KUKA KRL program: ps_ltc_geo_c2_bolha.src, ps_ltc_geo_c2_bolha.dat

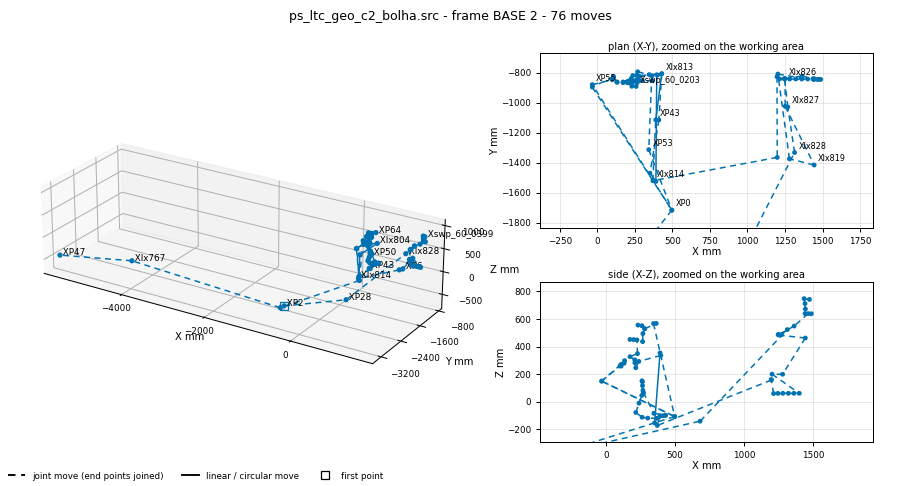
[picture p0: tool path of ps_ltc_geo_c2_bolha.src in frame BASE 2, 76 of 80 moves have a stored position in this frame; points joined in program order, loops and branches not executed]
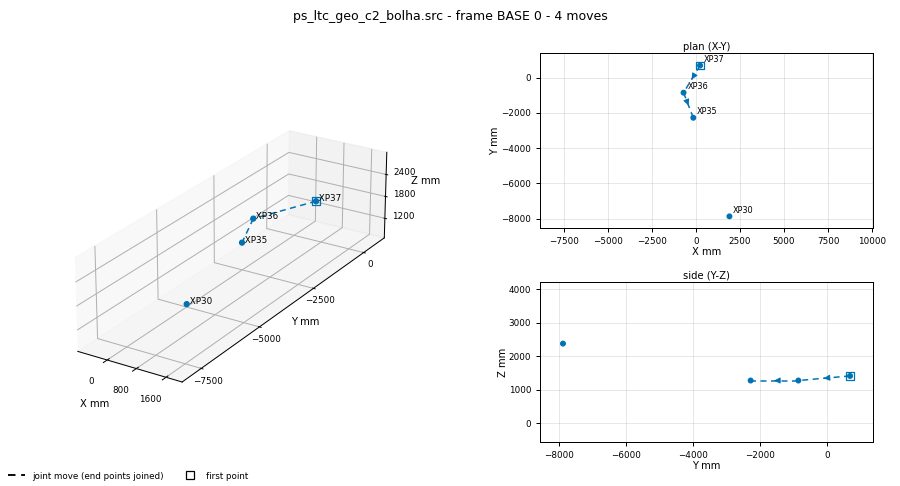
[picture p1: tool path of ps_ltc_geo_c2_bolha.src in frame BASE 0, 4 of 80 moves have a stored position in this frame; points joined in program order, loops and branches not executed]
--- ps_ltc_geo_c2_bolha.src ---
&ACCESS RVO1
&REL 3
&COMMENT GUN C2 geom Accelo
&PARAM DISKPATH = KRC:\R1\Program
DEF ps_ltc_geo_c2_bolha( )
;FOLD INI
;FOLD SPOTTECH INI
USERSPOT(#INIT)
;ENDFOLD (SPOTTECH INI)
;FOLD GRIPPERTECH INI
USER_GRP(0,DUMMY,DUMMY,GDEFAULT)
;ENDFOLD (GRIPPERTECH INI)
  ;FOLD USER INI
    ;Make your modifications here

  ;ENDFOLD (USER INI)
;ENDFOLD (INI)

; Caracterização dos meios de produção:
; Versão Atual:
; 12/07/2013 12:00 Name: P13.050-R3 CHANGES: Solda Geometria Accelo
; Pinça C2

chk_w2_wechs_ok ( )         ; CHECK C2

;FOLD PTP P37 CONT Vel=100 % PDAT38 Tool[2]:Gun C2 Base[2]:Accelo;%{PE}%R 8.2.20,%MKUKATPBASIS,%CMOVE,%VPTP,%P 1:PTP, 2:P37, 3:C_DIS, 5:100, 7:PDAT38
$BWDSTART=FALSE
PDAT_ACT=PPDAT38
FDAT_ACT=FP37
BAS(#PTP_PARAMS,100)
PTP XP37 C_DIS
;ENDFOLD

if MaxStandMenge (2) then
  MaxStandmengeErreicht (2)
endif

IF (NOT(GHOST())) THEN
if Elektrodenwechsel (2) then
  e_fraes2 ()
endif
ENDIF

;FOLD PTP P36 CONT Vel=100 % PDAT37 Tool[2]:Gun C2 Base[2]:Accelo;%{PE}%R 8.2.20,%MKUKATPBASIS,%CMOVE,%VPTP,%P 1:PTP, 2:P36, 3:C_DIS, 5:100, 7:PDAT37
$BWDSTART=FALSE
PDAT_ACT=PPDAT37
FDAT_ACT=FP36
BAS(#PTP_PARAMS,100)
PTP XP36 C_DIS
;ENDFOLD
;FOLD PTP P35 CONT Vel=100 % PDAT36 Tool[2]:Gun C2 Base[2]:Accelo;%{PE}%R 8.2.20,%MKUKATPBASIS,%CMOVE,%VPTP,%P 1:PTP, 2:P35, 3:C_DIS, 5:100, 7:PDAT36
$BWDSTART=FALSE
PDAT_ACT=PPDAT36
FDAT_ACT=FP35
BAS(#PTP_PARAMS,100)
PTP XP35 C_DIS
;ENDFOLD
;FOLD PTP P2 Vel=100 % PDAT2 Tool[2]:Gun C2 Base[2]:Accelo;%{PE}%R 8.2.20,%MKUKATPBASIS,%CMOVE,%VPTP,%P 1:PTP, 2:P2, 3:, 5:100, 7:PDAT2
$BWDSTART=FALSE
PDAT_ACT=PPDAT2
FDAT_ACT=FP2
BAS(#PTP_PARAMS,100)
PTP XP2
;ENDFOLD

;FOLD OUT 3339 'R3 Soldando' State=TRUE ;%{PE}%R 8.2.20,%MKUKATPBASIS,%COUT,%VOUTX,%P 2:3339, 3:R3 Soldando, 5:TRUE, 6:
$OUT[3339]=TRUE
;ENDFOLD
;FOLD WAIT FOR ( IN 3339 'Aguarda Lib. Soldar Geometria' );%{PE}%R 8.2.20,%MKUKATPBASIS,%CEXT_WAIT_FOR,%VEXT_WAIT_FOR,%P 2:, 4:, 5:$IN, 6:3339, 7:Aguarda Lib. Soldar Geometria, 9:
WAIT FOR  ( $IN[3339] )
;ENDFOLD
;FOLD OUT 3339 'R3 Soldando' State=FALSE ;%{PE}%R 8.2.20,%MKUKATPBASIS,%COUT,%VOUTX,%P 2:3339, 3:R3 Soldando, 5:FALSE, 6:
$OUT[3339]=FALSE
;ENDFOLD
;FOLD OUT 3348 'Fora area GEOBOX' State=FALSE ;%{PE}%R 8.2.20,%MKUKATPBASIS,%COUT,%VOUTX,%P 2:3348, 3:Fora area GEOBOX, 5:FALSE, 6:
$OUT[3348]=FALSE
;ENDFOLD

;FOLD Collision.Monitoring_AREA_1_On ;%{PE}%MKUKATPUSER
COLLSTOP( 7, 1 ) ;not Interrupt-Controlled
;ENDFOLD

;FOLD PTP P28 CONT Vel=100 % PDAT28 Tool[2]:Gun C2 Base[2]:Accelo;%{PE}%R 8.2.20,%MKUKATPBASIS,%CMOVE,%VPTP,%P 1:PTP, 2:P28, 3:C_DIS, 5:100, 7:PDAT28
$BWDSTART=FALSE
PDAT_ACT=PPDAT28
FDAT_ACT=FP28
BAS(#PTP_PARAMS,100)
PTP XP28 C_DIS
;ENDFOLD
;FOLD PTP lx828 CONT Vel=100 % P_OLP7 Tool[2]:Gun C2 Base[2]:Accelo;%{PE}%R 8.2.20,%MKUKATPBASIS,%CMOVE,%VPTP,%P 1:PTP, 2:lx828, 3:C_DIS, 5:100, 7:P_OLP7
$BWDSTART=FALSE
PDAT_ACT=PP_OLP7
FDAT_ACT=Flx828
BAS(#PTP_PARAMS,100)
PTP Xlx828 C_DIS
;ENDFOLD
;FOLD PTP lx827 CONT Vel=100 % P_OLP8 Tool[2]:Gun C2 Base[2]:Accelo;%{PE}%R 8.2.20,%MKUKATPBASIS,%CMOVE,%VPTP,%P 1:PTP, 2:lx827, 3:C_DIS, 5:100, 7:P_OLP8
$BWDSTART=FALSE
PDAT_ACT=PP_OLP8
FDAT_ACT=Flx827
BAS(#PTP_PARAMS,100)
PTP Xlx827 C_DIS
;ENDFOLD
;FOLD PTP lx826 CONT Vel=100 % P_OLP9 Tool[2]:Gun C2 Base[2]:Accelo;%{PE}%R 8.2.20,%MKUKATPBASIS,%CMOVE,%VPTP,%P 1:PTP, 2:lx826, 3:C_DIS, 5:100, 7:P_OLP9
$BWDSTART=FALSE
PDAT_ACT=PP_OLP9
FDAT_ACT=Flx826
BAS(#PTP_PARAMS,100)
PTP Xlx826 C_DIS
;ENDFOLD
;FOLD PTP P30 Vel=100 % PDAT30 Tool[2]:Gun C2 Base[0];%{PE}%R 8.2.20,%MKUKATPBASIS,%CMOVE,%VPTP,%P 1:PTP, 2:P30, 3:, 5:100, 7:PDAT30
$BWDSTART=FALSE
PDAT_ACT=PPDAT30
FDAT_ACT=FP30
BAS(#PTP_PARAMS,100)
PTP XP30
;ENDFOLD

;FOLD Collision.Monitoring_AREA_2_On ;%{PE}%MKUKATPUSER
COLLSTOP( 8, 1 ) ;not Interrupt-Controlled
;ENDFOLD

;FOLD ; swp_60_0399;%{PE}%R 5.4.33,%MKUKATPBASIS,%CCOMMENT,%VNORMAL,%P 2:swp_60_0399
;ENDFOLD
;FOLD PTP swp_60_0399 P_OLP10 SPOT Gun=2 RETR CLS PGNO1=110 ACTIVE=1 Tool[2]:Gun C2 Base[2]:Accelo;%{PE}%R 8.2.2,%MKUKATPSPOT,%CSPOT,%VPTP,%P 1:PTP, 2:swp_60_0399, 3:, 5:100, 7:P_OLP10, 10:2, 12:#FIRST, 14:#CLO, 16:151, 18:1, 20:1, 22:0, 24:1, 25:S_OLP1
$BWDSTART=FALSE
PDAT_ACT=PP_OLP10
FDAT_ACT=Fswp_60_0399
BAS(#PTP_PARAMS,PP_OLP10.VEL)
S_ACT.GUN=2
S_ACT.PAIR=SDEFAULT.PAIR
S_ACT.RETR=#CLO
S_ACT.CLO_TM=1
S_ACT.PGNO1=110
S_ACT.PGNO2=SDEFAULT.PGNO2
S_ACT.PRESS1=SDEFAULT.PRESS1
S_ACT.PRESS2=SDEFAULT.PRESS2
S_READY=FALSE
PTP Xswp_60_0399
USERSPOT(#SPOT, S_ACT)
WAIT FOR S_READY
;ENDFOLD

;FOLD PTP P41 CONT Vel=100 % PDAT42 Tool[2]:Gun C2 Base[2]:Accelo;%{PE}%R 8.2.20,%MKUKATPBASIS,%CMOVE,%VPTP,%P 1:PTP, 2:P41, 3:C_DIS, 5:100, 7:PDAT42
$BWDSTART=FALSE
PDAT_ACT=PPDAT42
FDAT_ACT=FP41
BAS(#PTP_PARAMS,100)
PTP XP41 C_DIS
;ENDFOLD


;FOLD ; swp_60_0397;%{PE}%R 8.2.20,%MKUKATPBASIS,%CCOMMENT,%VNORMAL,%P 2:swp_60_0397
;ENDFOLD
;FOLD PTP swp_60_0397 P_OLP15 SPOT Gun=2 RETR CLS PgNo1=145 ACTIVE=1 Tool[2]:Gun C2 Base[2]:Accelo;%{PE}%R 8.2.2,%MKUKATPSPOT,%CSPOT,%VPTP,%P 1:PTP, 2:swp_60_0397, 3:, 5:100, 7:P_OLP15, 10:2, 12:#FIRST, 14:#CLO, 16:145, 18:1, 20:1, 22:0, 24:1, 25:S_OLP2
$BWDSTART=FALSE
PDAT_ACT=PP_OLP15
FDAT_ACT=Fswp_60_0397
BAS(#PTP_PARAMS,PP_OLP15.VEL)
S_ACT.GUN=2
S_ACT.PAIR=SDEFAULT.PAIR
S_ACT.RETR=#CLO
S_ACT.CLO_TM=1
S_ACT.PGNO1=145
S_ACT.PGNO2=SDEFAULT.PGNO2
S_ACT.PRESS1=SDEFAULT.PRESS1
S_ACT.PRESS2=SDEFAULT.PRESS2
S_READY=FALSE
PTP Xswp_60_0397
USERSPOT(#SPOT, S_ACT)
WAIT FOR S_READY
;ENDFOLD

;FOLD ; swp_60_0395;%{PE}%R 5.4.33,%MKUKATPBASIS,%CCOMMENT,%VNORMAL,%P 2:swp_60_0395
;ENDFOLD
;FOLD PTP swp_60_0395 P_OLP12 SPOT Gun=2 RETR CLS PgNo1=111 ACTIVE=1 Tool[2]:Gun C2 Base[2]:Accelo;%{PE}%R 8.2.2,%MKUKATPSPOT,%CSPOT,%VPTP,%P 1:PTP, 2:swp_60_0395, 3:, 5:100, 7:P_OLP12, 10:2, 12:#FIRST, 14:#CLO, 16:111, 18:1, 20:1, 22:0, 24:1, 25:S_OLP2
$BWDSTART=FALSE
PDAT_ACT=PP_OLP12
FDAT_ACT=Fswp_60_0395
BAS(#PTP_PARAMS,PP_OLP12.VEL)
S_ACT.GUN=2
S_ACT.PAIR=SDEFAULT.PAIR
S_ACT.RETR=#CLO
S_ACT.CLO_TM=1
S_ACT.PGNO1=111
S_ACT.PGNO2=SDEFAULT.PGNO2
S_ACT.PRESS1=SDEFAULT.PRESS1
S_ACT.PRESS2=SDEFAULT.PRESS2
S_READY=FALSE
PTP Xswp_60_0395
USERSPOT(#SPOT, S_ACT)
WAIT FOR S_READY
;ENDFOLD

;FOLD PTP lx824 CONT Vel=100 % P_OLP13 Tool[2]:Gun C2 Base[2]:Accelo;%{PE}%R 8.2.20,%MKUKATPBASIS,%CMOVE,%VPTP,%P 1:PTP, 2:lx824, 3:C_DIS, 5:100, 7:P_OLP13
$BWDSTART=FALSE
PDAT_ACT=PP_OLP13
FDAT_ACT=Flx824
BAS(#PTP_PARAMS,100)
PTP Xlx824 C_DIS
;ENDFOLD


;FOLD ; swp_60_0391;%{PE}%R 8.2.20,%MKUKATPBASIS,%CCOMMENT,%VNORMAL,%P 2:swp_60_0391
;ENDFOLD
;FOLD PTP swp_60_0391 P_OLP17 SPOT Gun=2 RETR CLS PgNo1=146 ACTIVE=1 Tool[2]:Gun C2 Base[2]:Accelo;%{PE}%R 8.2.2,%MKUKATPSPOT,%CSPOT,%VPTP,%P 1:PTP, 2:swp_60_0391, 3:, 5:100, 7:P_OLP17, 10:2, 12:#FIRST, 14:#CLO, 16:146, 18:1, 20:1, 22:0, 24:1, 25:S_OLP3
$BWDSTART=FALSE
PDAT_ACT=PP_OLP17
FDAT_ACT=Fswp_60_0391
BAS(#PTP_PARAMS,PP_OLP17.VEL)
S_ACT.GUN=2
S_ACT.PAIR=SDEFAULT.PAIR
S_ACT.RETR=#CLO
S_ACT.CLO_TM=1
S_ACT.PGNO1=146
S_ACT.PGNO2=SDEFAULT.PGNO2
S_ACT.PRESS1=SDEFAULT.PRESS1
S_ACT.PRESS2=SDEFAULT.PRESS2
S_READY=FALSE
PTP Xswp_60_0391
USERSPOT(#SPOT, S_ACT)
WAIT FOR S_READY
;ENDFOLD

;FOLD ; swp_60_0393;%{PE}%R 5.4.33,%MKUKATPBASIS,%CCOMMENT,%VNORMAL,%P 2:swp_60_0393
;ENDFOLD
;FOLD PTP swp_60_0393 P_OLP14 SPOT Gun=2 RETR OPN PGNO1=112 ACTIVE=1 Tool[2]:Gun C2 Base[2]:Accelo;%{PE}%R 8.2.2,%MKUKATPSPOT,%CSPOT,%VPTP,%P 1:PTP, 2:swp_60_0393, 3:, 5:100, 7:P_OLP14, 10:2, 12:#FIRST, 14:#OPN, 16:153, 18:1, 20:1, 22:0, 24:1, 25:S_OLP3
$BWDSTART=FALSE
PDAT_ACT=PP_OLP14
FDAT_ACT=Fswp_60_0393
BAS(#PTP_PARAMS,PP_OLP14.VEL)
S_ACT.GUN=2
S_ACT.PAIR=SDEFAULT.PAIR
S_ACT.RETR=#OPN
S_ACT.CLO_TM=1
S_ACT.PGNO1=112
S_ACT.PGNO2=SDEFAULT.PGNO2
S_ACT.PRESS1=SDEFAULT.PRESS1
S_ACT.PRESS2=SDEFAULT.PRESS2
S_READY=FALSE
PTP Xswp_60_0393
USERSPOT(#SPOT, S_ACT)
WAIT FOR S_READY
;ENDFOLD

;FOLD PTP lx823 CONT Vel=100 % P_OLP16 Tool[2]:Gun C2 Base[2]:Accelo;%{PE}%R 8.2.20,%MKUKATPBASIS,%CMOVE,%VPTP,%P 1:PTP, 2:lx823, 3:C_DIS, 5:100, 7:P_OLP16
$BWDSTART=FALSE
PDAT_ACT=PP_OLP16
FDAT_ACT=Flx823
BAS(#PTP_PARAMS,100)
PTP Xlx823 C_DIS
;ENDFOLD
;FOLD PTP P42 Vel=100 % PDAT43 Tool[2]:Gun C2 Base[2]:Accelo;%{PE}%R 8.2.20,%MKUKATPBASIS,%CMOVE,%VPTP,%P 1:PTP, 2:P42, 3:, 5:100, 7:PDAT43
$BWDSTART=FALSE
PDAT_ACT=PPDAT43
FDAT_ACT=FP42
BAS(#PTP_PARAMS,100)
PTP XP42
;ENDFOLD
;FOLD PTP lx820 Vel=100 % P_OLP18 Tool[2]:Gun C2 Base[2]:Accelo;%{PE}%R 8.2.20,%MKUKATPBASIS,%CMOVE,%VPTP,%P 1:PTP, 2:lx820, 3:, 5:100, 7:P_OLP18
$BWDSTART=FALSE
PDAT_ACT=PP_OLP18
FDAT_ACT=Flx820
BAS(#PTP_PARAMS,100)
PTP Xlx820
;ENDFOLD

;FOLD Collision.Monitoring_AREA_2_Off . ;%{PE}%MKUKATPUSER
COLLSTOP( 8, 2+0 )
;ENDFOLD

;FOLD PTP lx819 CONT Vel=100 % P_OLP19 Tool[2]:Gun C2 Base[2]:Accelo;%{PE}%R 8.2.20,%MKUKATPBASIS,%CMOVE,%VPTP,%P 1:PTP, 2:lx819, 3:C_DIS, 5:100, 7:P_OLP19
$BWDSTART=FALSE
PDAT_ACT=PP_OLP19
FDAT_ACT=Flx819
BAS(#PTP_PARAMS,100)
PTP Xlx819 C_DIS
;ENDFOLD
;FOLD PTP P6 CONT Vel=100 % PDAT6 Tool[2]:Gun C2 Base[2]:Accelo;%{PE}%R 8.2.20,%MKUKATPBASIS,%CMOVE,%VPTP,%P 1:PTP, 2:P6, 3:C_DIS, 5:100, 7:PDAT6
$BWDSTART=FALSE
PDAT_ACT=PPDAT6
FDAT_ACT=FP6
BAS(#PTP_PARAMS,100)
PTP XP6 C_DIS
;ENDFOLD
;FOLD PTP P7 Vel=100 % PDAT7 Tool[2]:Gun C2 Base[2]:Accelo;%{PE}%R 8.2.20,%MKUKATPBASIS,%CMOVE,%VPTP,%P 1:PTP, 2:P7, 3:, 5:100, 7:PDAT7
$BWDSTART=FALSE
PDAT_ACT=PPDAT7
FDAT_ACT=FP7
BAS(#PTP_PARAMS,100)
PTP XP7
;ENDFOLD

;FOLD Collision.Monitoring_AREA_4_On ;%{PE}%MKUKATPUSER
COLLSTOP( 10, 1 ) ;not Interrupt-Controlled
;ENDFOLD

;FOLD ; swp_60_0341;%{PE}%R 8.2.20,%MKUKATPBASIS,%CCOMMENT,%VNORMAL,%P 2:swp_60_0341
;ENDFOLD
;FOLD PTP swp_60_0341 P_OLP21 SPOT Gun=2 RETR CLS PGNO1=113 ACTIVE=1 Tool[2]:Gun C2 Base[2]:Accelo;%{PE}%R 8.2.2,%MKUKATPSPOT,%CSPOT,%VPTP,%P 1:PTP, 2:swp_60_0341, 3:, 5:100, 7:P_OLP21, 10:2, 12:#FIRST, 14:#CLO, 16:154, 18:1, 20:1, 22:0, 24:1, 25:S_OLP4
$BWDSTART=FALSE
PDAT_ACT=PP_OLP21
FDAT_ACT=Fswp_60_0341
BAS(#PTP_PARAMS,PP_OLP21.VEL)
S_ACT.GUN=2
S_ACT.PAIR=SDEFAULT.PAIR
S_ACT.RETR=#CLO
S_ACT.CLO_TM=1
S_ACT.PGNO1=113
S_ACT.PGNO2=SDEFAULT.PGNO2
S_ACT.PRESS1=SDEFAULT.PRESS1
S_ACT.PRESS2=SDEFAULT.PRESS2
S_READY=FALSE
PTP Xswp_60_0341
USERSPOT(#SPOT, S_ACT)
WAIT FOR S_READY
;ENDFOLD

;FOLD ; swp_60_0339;%{PE}%R 8.2.20,%MKUKATPBASIS,%CCOMMENT,%VNORMAL,%P 2:swp_60_0339
;ENDFOLD
;FOLD PTP swp_60_0339 PDAT81 SPOT Gun=2 RETR CLS PGNO1=139 ACTIVE=1 Tool[2]:Gun C2 Base[2]:Accelo;%{PE}%R 8.2.2,%MKUKATPSPOT,%CSPOT,%VPTP,%P 1:PTP, 2:swp_60_0339, 3:, 5:100, 7:PDAT81, 10:2, 12:#FIRST, 14:#CLO, 16:180, 18:1, 20:0, 22:0, 24:1, 25:NORMAL
$BWDSTART=FALSE
PDAT_ACT=PPDAT81
FDAT_ACT=Fswp_60_0339
BAS(#PTP_PARAMS,PPDAT81.VEL)
S_ACT.GUN=2
S_ACT.PAIR=SDEFAULT.PAIR
S_ACT.RETR=#CLO
S_ACT.CLO_TM=1
S_ACT.PGNO1=139
S_ACT.PGNO2=SDEFAULT.PGNO2
S_ACT.PRESS1=SDEFAULT.PRESS1
S_ACT.PRESS2=SDEFAULT.PRESS2
S_READY=FALSE
PTP Xswp_60_0339
USERSPOT(#SPOT, S_ACT)
WAIT FOR S_READY
;ENDFOLD

;FOLD ; swp_60_0337;%{PE}%R 8.2.20,%MKUKATPBASIS,%CCOMMENT,%VNORMAL,%P 2:swp_60_0337
;ENDFOLD
;FOLD PTP swp_60_0337 PDAT82 SPOT Gun=2 RETR CLS PGNO1=140 ACTIVE=1 Tool[2]:Gun C2 Base[2]:Accelo;%{PE}%R 8.2.2,%MKUKATPSPOT,%CSPOT,%VPTP,%P 1:PTP, 2:swp_60_0337, 3:, 5:100, 7:PDAT82, 10:2, 12:#FIRST, 14:#CLO, 16:181, 18:1, 20:0, 22:0, 24:1, 25:NORMAL
$BWDSTART=FALSE
PDAT_ACT=PPDAT82
FDAT_ACT=Fswp_60_0337
BAS(#PTP_PARAMS,PPDAT82.VEL)
S_ACT.GUN=2
S_ACT.PAIR=SDEFAULT.PAIR
S_ACT.RETR=#CLO
S_ACT.CLO_TM=1
S_ACT.PGNO1=140
S_ACT.PGNO2=SDEFAULT.PGNO2
S_ACT.PRESS1=SDEFAULT.PRESS1
S_ACT.PRESS2=SDEFAULT.PRESS2
S_READY=FALSE
PTP Xswp_60_0337
USERSPOT(#SPOT, S_ACT)
WAIT FOR S_READY
;ENDFOLD

;FOLD ; swp_60_0335;%{PE}%R 8.2.20,%MKUKATPBASIS,%CCOMMENT,%VNORMAL,%P 2:swp_60_0335
;ENDFOLD
;FOLD PTP swp_60_0335 PDAT84 SPOT Gun=2 RETR CLS PGNO1=141 ACTIVE=1 Tool[2]:Gun C2 Base[2]:Accelo;%{PE}%R 8.2.2,%MKUKATPSPOT,%CSPOT,%VPTP,%P 1:PTP, 2:swp_60_0335, 3:, 5:100, 7:PDAT84, 10:2, 12:#FIRST, 14:#CLO, 16:182, 18:1, 20:0, 22:0, 24:1, 25:NORMAL
$BWDSTART=FALSE
PDAT_ACT=PPDAT84
FDAT_ACT=Fswp_60_0335
BAS(#PTP_PARAMS,PPDAT84.VEL)
S_ACT.GUN=2
S_ACT.PAIR=SDEFAULT.PAIR
S_ACT.RETR=#CLO
S_ACT.CLO_TM=1
S_ACT.PGNO1=141
S_ACT.PGNO2=SDEFAULT.PGNO2
S_ACT.PRESS1=SDEFAULT.PRESS1
S_ACT.PRESS2=SDEFAULT.PRESS2
S_READY=FALSE
PTP Xswp_60_0335
USERSPOT(#SPOT, S_ACT)
WAIT FOR S_READY
;ENDFOLD

;FOLD ; swp_60_0333;%{PE}%R 8.2.20,%MKUKATPBASIS,%CCOMMENT,%VNORMAL,%P 2:swp_60_0333
;ENDFOLD
;FOLD PTP swp_60_0333 PDAT83 SPOT Gun=2 RETR CLS PGNO1=142 ACTIVE=1 Tool[2]:Gun C2 Base[2]:Accelo;%{PE}%R 8.2.2,%MKUKATPSPOT,%CSPOT,%VPTP,%P 1:PTP, 2:swp_60_0333, 3:, 5:100, 7:PDAT83, 10:2, 12:#FIRST, 14:#CLO, 16:183, 18:1, 20:0, 22:0, 24:1, 25:NORMAL
$BWDSTART=FALSE
PDAT_ACT=PPDAT83
FDAT_ACT=Fswp_60_0333
BAS(#PTP_PARAMS,PPDAT83.VEL)
S_ACT.GUN=2
S_ACT.PAIR=SDEFAULT.PAIR
S_ACT.RETR=#CLO
S_ACT.CLO_TM=1
S_ACT.PGNO1=142
S_ACT.PGNO2=SDEFAULT.PGNO2
S_ACT.PRESS1=SDEFAULT.PRESS1
S_ACT.PRESS2=SDEFAULT.PRESS2
S_READY=FALSE
PTP Xswp_60_0333
USERSPOT(#SPOT, S_ACT)
WAIT FOR S_READY
;ENDFOLD

;FOLD ; swp_60_0331;%{PE}%R 8.2.20,%MKUKATPBASIS,%CCOMMENT,%VNORMAL,%P 2:swp_60_0331
;ENDFOLD
;FOLD PTP swp_60_0331 P_OLP22 SPOT Gun=2 RETR OPN PGNO1=114 ACTIVE=1 Tool[2]:Gun C2 Base[2]:Accelo;%{PE}%R 8.2.2,%MKUKATPSPOT,%CSPOT,%VPTP,%P 1:PTP, 2:swp_60_0331, 3:, 5:100, 7:P_OLP22, 10:2, 12:#FIRST, 14:#OPN, 16:155, 18:1, 20:1, 22:0, 24:1, 25:S_OLP5
$BWDSTART=FALSE
PDAT_ACT=PP_OLP22
FDAT_ACT=Fswp_60_0331
BAS(#PTP_PARAMS,PP_OLP22.VEL)
S_ACT.GUN=2
S_ACT.PAIR=SDEFAULT.PAIR
S_ACT.RETR=#OPN
S_ACT.CLO_TM=1
S_ACT.PGNO1=114
S_ACT.PGNO2=SDEFAULT.PGNO2
S_ACT.PRESS1=SDEFAULT.PRESS1
S_ACT.PRESS2=SDEFAULT.PRESS2
S_READY=FALSE
PTP Xswp_60_0331
USERSPOT(#SPOT, S_ACT)
WAIT FOR S_READY
;ENDFOLD

;FOLD PTP lx815 Vel=100 % P_OLP23 Tool[2]:Gun C2 Base[2]:Accelo;%{PE}%R 8.2.20,%MKUKATPBASIS,%CMOVE,%VPTP,%P 1:PTP, 2:lx815, 3:, 5:100, 7:P_OLP23
$BWDSTART=FALSE
PDAT_ACT=PP_OLP23
FDAT_ACT=Flx815
BAS(#PTP_PARAMS,100)
PTP Xlx815
;ENDFOLD

;FOLD Collision.Monitoring_AREA_4_Off . ;%{PE}%MKUKATPUSER
COLLSTOP( 10, 2+0 )
;ENDFOLD

;FOLD PTP lx816 CONT Vel=100 % P_OLP24 Tool[2]:Gun C2 Base[2]:Accelo;%{PE}%R 8.2.20,%MKUKATPBASIS,%CMOVE,%VPTP,%P 1:PTP, 2:lx816, 3:C_DIS, 5:100, 7:P_OLP24
$BWDSTART=FALSE
PDAT_ACT=PP_OLP24
FDAT_ACT=Flx816
BAS(#PTP_PARAMS,100)
PTP Xlx816 C_DIS
;ENDFOLD
;FOLD PTP lx814 Vel=100 % PDAT35 Tool[2]:Gun C2 Base[2]:Accelo;%{PE}%R 8.2.20,%MKUKATPBASIS,%CMOVE,%VPTP,%P 1:PTP, 2:lx814, 3:, 5:100, 7:PDAT35
$BWDSTART=FALSE
PDAT_ACT=PPDAT35
FDAT_ACT=Flx814
BAS(#PTP_PARAMS,100)
PTP Xlx814
;ENDFOLD

;FOLD Collision.Monitoring_AREA_3_On ;%{PE}%MKUKATPUSER
COLLSTOP( 9, 1 ) ;not Interrupt-Controlled
;ENDFOLD
;FOLD Collision.Monitoring_AREA_1_Off . ;%{PE}%MKUKATPUSER
COLLSTOP( 7, 2+0 )
;ENDFOLD

;FOLD PTP P43 CONT Vel=100 % PDAT85 Tool[2]:Gun C2 Base[2]:Accelo;%{PE}%R 8.2.20,%MKUKATPBASIS,%CMOVE,%VPTP,%P 1:PTP, 2:P43, 3:C_DIS, 5:100, 7:PDAT85
$BWDSTART=FALSE
PDAT_ACT=PPDAT85
FDAT_ACT=FP43
BAS(#PTP_PARAMS,100)
PTP XP43 C_DIS
;ENDFOLD

;FOLD LIN lx813 CONT Vel=1 m/s CPDAT5 Tool[2]:Gun C2 Base[2]:Accelo;%{PE}%R 8.2.20,%MKUKATPBASIS,%CMOVE,%VLIN,%P 1:LIN, 2:lx813, 3:C_DIS C_DIS, 5:1, 7:CPDAT5
$BWDSTART=FALSE
LDAT_ACT=LCPDAT5
FDAT_ACT=Flx813
BAS(#CP_PARAMS,1)
LIN Xlx813 C_DIS C_DIS
;ENDFOLD

;FOLD ; swp_60_0259;%{PE}%R 8.2.20,%MKUKATPBASIS,%CCOMMENT,%VNORMAL,%P 2:swp_60_0259
;ENDFOLD
;FOLD PTP swp_60_0259 PDAT55 SPOT Gun=2 RETR CLS PGNO1=96 ACTIVE=1 Tool[2]:Gun C2 Base[2]:Accelo;%{PE}%R 8.2.2,%MKUKATPSPOT,%CSPOT,%VPTP,%P 1:PTP, 2:swp_60_0259, 3:, 5:100, 7:PDAT55, 10:2, 12:#FIRST, 14:#CLO, 16:137, 18:1, 20:0, 22:0, 24:1, 25:NORMAL
$BWDSTART=FALSE
PDAT_ACT=PPDAT55
FDAT_ACT=Fswp_60_0259
BAS(#PTP_PARAMS,PPDAT55.VEL)
S_ACT.GUN=2
S_ACT.PAIR=SDEFAULT.PAIR
S_ACT.RETR=#CLO
S_ACT.CLO_TM=1
S_ACT.PGNO1=96
S_ACT.PGNO2=SDEFAULT.PGNO2
S_ACT.PRESS1=SDEFAULT.PRESS1
S_ACT.PRESS2=SDEFAULT.PRESS2
S_READY=FALSE
PTP Xswp_60_0259
USERSPOT(#SPOT, S_ACT)
WAIT FOR S_READY
;ENDFOLD

;FOLD ; swp_60_0255;%{PE}%R 5.4.33,%MKUKATPBASIS,%CCOMMENT,%VNORMAL,%P 2:swp_60_0255
;ENDFOLD
;FOLD PTP swp_60_0255 P_OLP30 SPOT Gun=2 RETR CLS PGNO1=115 ACTIVE=1 Tool[2]:Gun C2 Base[2]:Accelo;%{PE}%R 8.2.2,%MKUKATPSPOT,%CSPOT,%VPTP,%P 1:PTP, 2:swp_60_0255, 3:, 5:100, 7:P_OLP30, 10:2, 12:#FIRST, 14:#CLO, 16:156, 18:1, 20:1, 22:0, 24:1, 25:S_OLP6
$BWDSTART=FALSE
PDAT_ACT=PP_OLP30
FDAT_ACT=Fswp_60_0255
BAS(#PTP_PARAMS,PP_OLP30.VEL)
S_ACT.GUN=2
S_ACT.PAIR=SDEFAULT.PAIR
S_ACT.RETR=#CLO
S_ACT.CLO_TM=1
S_ACT.PGNO1=115
S_ACT.PGNO2=SDEFAULT.PGNO2
S_ACT.PRESS1=SDEFAULT.PRESS1
S_ACT.PRESS2=SDEFAULT.PRESS2
S_READY=FALSE
PTP Xswp_60_0255
USERSPOT(#SPOT, S_ACT)
WAIT FOR S_READY
;ENDFOLD

;FOLD ; swp_60_0253;%{PE}%R 8.2.20,%MKUKATPBASIS,%CCOMMENT,%VNORMAL,%P 2:swp_60_0253
;ENDFOLD
;FOLD PTP swp_60_0253 PDAT56 SPOT Gun=2 RETR CLS PGNO1=94 ACTIVE=1 Tool[2]:Gun C2 Base[2]:Accelo;%{PE}%R 8.2.2,%MKUKATPSPOT,%CSPOT,%VPTP,%P 1:PTP, 2:swp_60_0253, 3:, 5:100, 7:PDAT56, 10:2, 12:#FIRST, 14:#CLO, 16:135, 18:1, 20:0, 22:0, 24:1, 25:NORMAL
$BWDSTART=FALSE
PDAT_ACT=PPDAT56
FDAT_ACT=Fswp_60_0253
BAS(#PTP_PARAMS,PPDAT56.VEL)
S_ACT.GUN=2
S_ACT.PAIR=SDEFAULT.PAIR
S_ACT.RETR=#CLO
S_ACT.CLO_TM=1
S_ACT.PGNO1=94
S_ACT.PGNO2=SDEFAULT.PGNO2
S_ACT.PRESS1=SDEFAULT.PRESS1
S_ACT.PRESS2=SDEFAULT.PRESS2
S_READY=FALSE
PTP Xswp_60_0253
USERSPOT(#SPOT, S_ACT)
WAIT FOR S_READY
;ENDFOLD

;FOLD ; swp_60_0249;%{PE}%R 8.2.20,%MKUKATPBASIS,%CCOMMENT,%VNORMAL,%P 2:swp_60_0249
;ENDFOLD
;FOLD PTP swp_60_0249 PDAT57 SPOT Gun=2 RETR CLS PGNO1=92 ACTIVE=1 Tool[2]:Gun C2 Base[2]:Accelo;%{PE}%R 8.2.2,%MKUKATPSPOT,%CSPOT,%VPTP,%P 1:PTP, 2:swp_60_0249, 3:, 5:100, 7:PDAT57, 10:2, 12:#FIRST, 14:#CLO, 16:133, 18:1, 20:0, 22:0, 24:1, 25:NORMAL
$BWDSTART=FALSE
PDAT_ACT=PPDAT57
FDAT_ACT=Fswp_60_0249
BAS(#PTP_PARAMS,PPDAT57.VEL)
S_ACT.GUN=2
S_ACT.PAIR=SDEFAULT.PAIR
S_ACT.RETR=#CLO
S_ACT.CLO_TM=1
S_ACT.PGNO1=92
S_ACT.PGNO2=SDEFAULT.PGNO2
S_ACT.PRESS1=SDEFAULT.PRESS1
S_ACT.PRESS2=SDEFAULT.PRESS2
S_READY=FALSE
PTP Xswp_60_0249
USERSPOT(#SPOT, S_ACT)
WAIT FOR S_READY
;ENDFOLD

;FOLD ; swp_60_0245;%{PE}%R 5.4.33,%MKUKATPBASIS,%CCOMMENT,%VNORMAL,%P 2:swp_60_0245
;ENDFOLD
;FOLD PTP swp_60_0245 P_OLP31 SPOT Gun=2 RETR CLS PGNO1=116 ACTIVE=1 Tool[2]:Gun C2 Base[2]:Accelo;%{PE}%R 8.2.2,%MKUKATPSPOT,%CSPOT,%VPTP,%P 1:PTP, 2:swp_60_0245, 3:, 5:100, 7:P_OLP31, 10:2, 12:#FIRST, 14:#CLO, 16:157, 18:1, 20:1, 22:0, 24:1, 25:S_OLP7
$BWDSTART=FALSE
PDAT_ACT=PP_OLP31
FDAT_ACT=Fswp_60_0245
BAS(#PTP_PARAMS,PP_OLP31.VEL)
S_ACT.GUN=2
S_ACT.PAIR=SDEFAULT.PAIR
S_ACT.RETR=#CLO
S_ACT.CLO_TM=1
S_ACT.PGNO1=116
S_ACT.PGNO2=SDEFAULT.PGNO2
S_ACT.PRESS1=SDEFAULT.PRESS1
S_ACT.PRESS2=SDEFAULT.PRESS2
S_READY=FALSE
PTP Xswp_60_0245
USERSPOT(#SPOT, S_ACT)
WAIT FOR S_READY
;ENDFOLD

;FOLD ; swp_60_0241;%{PE}%R 8.2.20,%MKUKATPBASIS,%CCOMMENT,%VNORMAL,%P 2:swp_60_0241
;ENDFOLD
;FOLD PTP swp_60_0241 PDAT58 SPOT Gun=2 RETR CLS PGNO1=89 ACTIVE=1 Tool[2]:Gun C2 Base[2]:Accelo;%{PE}%R 8.2.2,%MKUKATPSPOT,%CSPOT,%VPTP,%P 1:PTP, 2:swp_60_0241, 3:, 5:100, 7:PDAT58, 10:2, 12:#FIRST, 14:#CLO, 16:130, 18:1, 20:0, 22:0, 24:1, 25:NORMAL
$BWDSTART=FALSE
PDAT_ACT=PPDAT58
FDAT_ACT=Fswp_60_0241
BAS(#PTP_PARAMS,PPDAT58.VEL)
S_ACT.GUN=2
S_ACT.PAIR=SDEFAULT.PAIR
S_ACT.RETR=#CLO
S_ACT.CLO_TM=1
S_ACT.PGNO1=89
S_ACT.PGNO2=SDEFAULT.PGNO2
S_ACT.PRESS1=SDEFAULT.PRESS1
S_ACT.PRESS2=SDEFAULT.PRESS2
S_READY=FALSE
PTP Xswp_60_0241
USERSPOT(#SPOT, S_ACT)
WAIT FOR S_READY
;ENDFOLD

;FOLD PTP P50 CONT Vel=100 % PDAT59 Tool[2]:Gun C2 Base[2]:Accelo;%{PE}%R 8.2.20,%MKUKATPBASIS,%CMOVE,%VPTP,%P 1:PTP, 2:P50, 3:C_DIS, 5:100, 7:PDAT59
$BWDSTART=FALSE
PDAT_ACT=PPDAT59
FDAT_ACT=FP50
BAS(#PTP_PARAMS,100)
PTP XP50 C_DIS
;ENDFOLD

;FOLD ; swp_60_0239;%{PE}%R 8.2.20,%MKUKATPBASIS,%CCOMMENT,%VNORMAL,%P 2:swp_60_0239
;ENDFOLD
;FOLD PTP swp_60_0239 PDAT60 SPOT Gun=2 RETR CLS PGNO1=88 ACTIVE=1 Tool[2]:Gun C2 Base[2]:Accelo;%{PE}%R 8.2.2,%MKUKATPSPOT,%CSPOT,%VPTP,%P 1:PTP, 2:swp_60_0239, 3:, 5:100, 7:PDAT60, 10:2, 12:#FIRST, 14:#CLO, 16:129, 18:1, 20:0, 22:0, 24:1, 25:NORMAL
$BWDSTART=FALSE
PDAT_ACT=PPDAT60
FDAT_ACT=Fswp_60_0239
BAS(#PTP_PARAMS,PPDAT60.VEL)
S_ACT.GUN=2
S_ACT.PAIR=SDEFAULT.PAIR
S_ACT.RETR=#CLO
S_ACT.CLO_TM=1
S_ACT.PGNO1=88
S_ACT.PGNO2=SDEFAULT.PGNO2
S_ACT.PRESS1=SDEFAULT.PRESS1
S_ACT.PRESS2=SDEFAULT.PRESS2
S_READY=FALSE
PTP Xswp_60_0239
USERSPOT(#SPOT, S_ACT)
WAIT FOR S_READY
;ENDFOLD

;FOLD ; swp_60_0237;%{PE}%R 8.2.20,%MKUKATPBASIS,%CCOMMENT,%VNORMAL,%P 2:swp_60_0237
;ENDFOLD
;FOLD PTP swp_60_0237 PDAT61 SPOT Gun=2 RETR CLS PGNO1=87 ACTIVE=1 Tool[2]:Gun C2 Base[2]:Accelo;%{PE}%R 8.2.2,%MKUKATPSPOT,%CSPOT,%VPTP,%P 1:PTP, 2:swp_60_0237, 3:, 5:100, 7:PDAT61, 10:2, 12:#FIRST, 14:#CLO, 16:128, 18:1, 20:0, 22:0, 24:1, 25:NORMAL
$BWDSTART=FALSE
PDAT_ACT=PPDAT61
FDAT_ACT=Fswp_60_0237
BAS(#PTP_PARAMS,PPDAT61.VEL)
S_ACT.GUN=2
S_ACT.PAIR=SDEFAULT.PAIR
S_ACT.RETR=#CLO
S_ACT.CLO_TM=1
S_ACT.PGNO1=87
S_ACT.PGNO2=SDEFAULT.PGNO2
S_ACT.PRESS1=SDEFAULT.PRESS1
S_ACT.PRESS2=SDEFAULT.PRESS2
S_READY=FALSE
PTP Xswp_60_0237
USERSPOT(#SPOT, S_ACT)
WAIT FOR S_READY
;ENDFOLD

;FOLD PTP P11 CONT Vel=50 % PDAT11 Tool[2]:Gun C2 Base[2]:Accelo;%{PE}%R 8.2.20,%MKUKATPBASIS,%CMOVE,%VPTP,%P 1:PTP, 2:P11, 3:C_DIS, 5:50, 7:PDAT11
$BWDSTART=FALSE
PDAT_ACT=PPDAT11
FDAT_ACT=FP11
BAS(#PTP_PARAMS,50)
PTP XP11 C_DIS
;ENDFOLD

;FOLD ; swp_60_0235;%{PE}%R 5.4.33,%MKUKATPBASIS,%CCOMMENT,%VNORMAL,%P 2:swp_60_0235
;ENDFOLD
;FOLD PTP swp_60_0235 P_OLP33 SPOT Gun=2 RETR OPN PGNO1=117 ACTIVE=1 Tool[2]:Gun C2 Base[2]:Accelo;%{PE}%R 8.2.2,%MKUKATPSPOT,%CSPOT,%VPTP,%P 1:PTP, 2:swp_60_0235, 3:, 5:100, 7:P_OLP33, 10:2, 12:#FIRST, 14:#OPN, 16:158, 18:1, 20:1, 22:0, 24:1, 25:S_OLP8
$BWDSTART=FALSE
PDAT_ACT=PP_OLP33
FDAT_ACT=Fswp_60_0235
BAS(#PTP_PARAMS,PP_OLP33.VEL)
S_ACT.GUN=2
S_ACT.PAIR=SDEFAULT.PAIR
S_ACT.RETR=#OPN
S_ACT.CLO_TM=1
S_ACT.PGNO1=117
S_ACT.PGNO2=SDEFAULT.PGNO2
S_ACT.PRESS1=SDEFAULT.PRESS1
S_ACT.PRESS2=SDEFAULT.PRESS2
S_READY=FALSE
PTP Xswp_60_0235
USERSPOT(#SPOT, S_ACT)
WAIT FOR S_READY
;ENDFOLD

;FOLD PTP lx798 CONT Vel=100 % P_OLP34 Tool[2]:Gun C2 Base[2]:Accelo;%{PE}%R 8.2.20,%MKUKATPBASIS,%CMOVE,%VPTP,%P 1:PTP, 2:lx798, 3:C_DIS, 5:100, 7:P_OLP34
$BWDSTART=FALSE
PDAT_ACT=PP_OLP34
FDAT_ACT=Flx798
BAS(#PTP_PARAMS,100)
PTP Xlx798 C_DIS
;ENDFOLD
;FOLD PTP lx799 CONT Vel=100 % P_OLP35 Tool[2]:Gun C2 Base[2]:Accelo;%{PE}%R 8.2.20,%MKUKATPBASIS,%CMOVE,%VPTP,%P 1:PTP, 2:lx799, 3:C_DIS, 5:100, 7:P_OLP35
$BWDSTART=FALSE
PDAT_ACT=PP_OLP35
FDAT_ACT=Flx799
BAS(#PTP_PARAMS,100)
PTP Xlx799 C_DIS
;ENDFOLD

;FOLD LIN lx800 CONT Vel=1 m/s CPDAT8 Tool[2]:Gun C2 Base[2]:Accelo;%{PE}%R 8.2.20,%MKUKATPBASIS,%CMOVE,%VLIN,%P 1:LIN, 2:lx800, 3:C_DIS C_DIS, 5:1, 7:CPDAT8
$BWDSTART=FALSE
LDAT_ACT=LCPDAT8
FDAT_ACT=Flx800
BAS(#CP_PARAMS,1)
LIN Xlx800 C_DIS C_DIS
;ENDFOLD

;FOLD PTP lx802 CONT Vel=100 % P_OLP37 Tool[2]:Gun C2 Base[2]:Accelo;%{PE}%R 8.2.20,%MKUKATPBASIS,%CMOVE,%VPTP,%P 1:PTP, 2:lx802, 3:C_DIS, 5:100, 7:P_OLP37
$BWDSTART=FALSE
PDAT_ACT=PP_OLP37
FDAT_ACT=Flx802
BAS(#PTP_PARAMS,100)
PTP Xlx802 C_DIS
;ENDFOLD
;FOLD PTP lx801 CONT Vel=100 % P_OLP38 Tool[2]:Gun C2 Base[2]:Accelo;%{PE}%R 8.2.20,%MKUKATPBASIS,%CMOVE,%VPTP,%P 1:PTP, 2:lx801, 3:C_DIS, 5:100, 7:P_OLP38
$BWDSTART=FALSE
PDAT_ACT=PP_OLP38
FDAT_ACT=Flx801
BAS(#PTP_PARAMS,100)
PTP Xlx801 C_DIS
;ENDFOLD

;FOLD LIN P62 CONT Vel=1.5 m/s CPDAT11 Tool[2]:Gun C2 Base[2]:Accelo;%{PE}%R 8.2.20,%MKUKATPBASIS,%CMOVE,%VLIN,%P 1:LIN, 2:P62, 3:C_DIS C_DIS, 5:1.5, 7:CPDAT11
$BWDSTART=FALSE
LDAT_ACT=LCPDAT11
FDAT_ACT=FP62
BAS(#CP_PARAMS,1.5)
LIN XP62 C_DIS C_DIS
;ENDFOLD
;FOLD LIN lx804 CONT Vel=1 m/s CPDAT1 Tool[2]:Gun C2 Base[2]:Accelo;%{PE}%R 8.2.20,%MKUKATPBASIS,%CMOVE,%VLIN,%P 1:LIN, 2:lx804, 3:C_DIS C_DIS, 5:1, 7:CPDAT1
$BWDSTART=FALSE
LDAT_ACT=LCPDAT1
FDAT_ACT=Flx804
BAS(#CP_PARAMS,1)
LIN Xlx804 C_DIS C_DIS
;ENDFOLD

;FOLD PTP lx803 CONT Vel=100 % P_OLP45 Tool[2]:Gun C2 Base[2]:Accelo;%{PE}%R 8.2.20,%MKUKATPBASIS,%CMOVE,%VPTP,%P 1:PTP, 2:lx803, 3:C_DIS, 5:100, 7:P_OLP45
$BWDSTART=FALSE
PDAT_ACT=PP_OLP45
FDAT_ACT=Flx803
BAS(#PTP_PARAMS,100)
PTP Xlx803 C_DIS
;ENDFOLD

;FOLD ; swp_60_0229;%{PE}%R 5.4.33,%MKUKATPBASIS,%CCOMMENT,%VNORMAL,%P 2:swp_60_0229
;ENDFOLD
;FOLD PTP swp_60_0229 P_OLP46 SPOT Gun=2 RETR CLS PGNO1=118 ACTIVE=1 Tool[2]:Gun C2 Base[2]:Accelo;%{PE}%R 8.2.2,%MKUKATPSPOT,%CSPOT,%VPTP,%P 1:PTP, 2:swp_60_0229, 3:, 5:100, 7:P_OLP46, 10:2, 12:#FIRST, 14:#CLO, 16:159, 18:1, 20:1, 22:0, 24:1, 25:S_OLP9
$BWDSTART=FALSE
PDAT_ACT=PP_OLP46
FDAT_ACT=Fswp_60_0229
BAS(#PTP_PARAMS,PP_OLP46.VEL)
S_ACT.GUN=2
S_ACT.PAIR=SDEFAULT.PAIR
S_ACT.RETR=#CLO
S_ACT.CLO_TM=1
S_ACT.PGNO1=118
S_ACT.PGNO2=SDEFAULT.PGNO2
S_ACT.PRESS1=SDEFAULT.PRESS1
S_ACT.PRESS2=SDEFAULT.PRESS2
S_READY=FALSE
PTP Xswp_60_0229
USERSPOT(#SPOT, S_ACT)
WAIT FOR S_READY
;ENDFOLD

;FOLD ; swp_60_0225;%{PE}%R 5.4.33,%MKUKATPBASIS,%CCOMMENT,%VNORMAL,%P 2:swp_60_0225
;ENDFOLD
;FOLD PTP swp_60_0225 P_OLP47 SPOT Gun=2 RETR CLS PGNO1=119 ACTIVE=1 Tool[2]:Gun C2 Base[2]:Accelo;%{PE}%R 8.2.2,%MKUKATPSPOT,%CSPOT,%VPTP,%P 1:PTP, 2:swp_60_0225, 3:, 5:100, 7:P_OLP47, 10:2, 12:#FIRST, 14:#CLO, 16:160, 18:1, 20:1, 22:0, 24:1, 25:S_OLP10
$BWDSTART=FALSE
PDAT_ACT=PP_OLP47
FDAT_ACT=Fswp_60_0225
BAS(#PTP_PARAMS,PP_OLP47.VEL)
S_ACT.GUN=2
S_ACT.PAIR=SDEFAULT.PAIR
S_ACT.RETR=#CLO
S_ACT.CLO_TM=1
S_ACT.PGNO1=119
S_ACT.PGNO2=SDEFAULT.PGNO2
S_ACT.PRESS1=SDEFAULT.PRESS1
S_ACT.PRESS2=SDEFAULT.PRESS2
S_READY=FALSE
PTP Xswp_60_0225
USERSPOT(#SPOT, S_ACT)
WAIT FOR S_READY
;ENDFOLD

;FOLD PTP PS01010021 PDAT86 RETR OPN Gun=2 Tool[2]:Gun C2 Base[2]:Accelo;%{PE}%R 8.2.2,%MKUKATPSPOT,%CRETR,%VPTP,%P 1:PTP, 2:PS01010021, 3:, 5:100, 7:PDAT86, 9:#OPN, 11:2, 13:#FIRST
$BWDSTART=FALSE
PDAT_ACT=PPDAT86
FDAT_ACT=FPS01010021
BAS(#PTP_PARAMS,PPDAT86.VEL)
S_ACT.GUN=2
S_ACT.PAIR=#FIRST
S_ACT.RETR=#OPN
S_READY=FALSE
PTP XPS01010021
USERSPOT(#RETR, S_ACT)
WAIT FOR S_READY
;ENDFOLD

;FOLD ; swp_60_0221;%{PE}%R 5.4.33,%MKUKATPBASIS,%CCOMMENT,%VNORMAL,%P 2:swp_60_0221
;ENDFOLD
;FOLD PTP swp_60_0221 P_OLP49 SPOT Gun=2 RETR OPN PGNO1=120 ACTIVE=1 Tool[2]:Gun C2 Base[2]:Accelo;%{PE}%R 8.2.2,%MKUKATPSPOT,%CSPOT,%VPTP,%P 1:PTP, 2:swp_60_0221, 3:, 5:100, 7:P_OLP49, 10:2, 12:#FIRST, 14:#OPN, 16:161, 18:1, 20:1, 22:0, 24:1, 25:S_OLP11
$BWDSTART=FALSE
PDAT_ACT=PP_OLP49
FDAT_ACT=Fswp_60_0221
BAS(#PTP_PARAMS,PP_OLP49.VEL)
S_ACT.GUN=2
S_ACT.PAIR=SDEFAULT.PAIR
S_ACT.RETR=#OPN
S_ACT.CLO_TM=1
S_ACT.PGNO1=120
S_ACT.PGNO2=SDEFAULT.PGNO2
S_ACT.PRESS1=SDEFAULT.PRESS1
S_ACT.PRESS2=SDEFAULT.PRESS2
S_READY=FALSE
PTP Xswp_60_0221
USERSPOT(#SPOT, S_ACT)
WAIT FOR S_READY
;ENDFOLD

;FOLD PTP lx795 CONT Vel=100 % P_OLP50 Tool[2]:Gun C2 Base[2]:Accelo;%{PE}%R 8.2.20,%MKUKATPBASIS,%CMOVE,%VPTP,%P 1:PTP, 2:lx795, 3:C_DIS, 5:100, 7:P_OLP50
$BWDSTART=FALSE
PDAT_ACT=PP_OLP50
FDAT_ACT=Flx795
BAS(#PTP_PARAMS,100)
PTP Xlx795 C_DIS
;ENDFOLD

;FOLD ; swp_60_0207;%{PE}%R 8.2.20,%MKUKATPBASIS,%CCOMMENT,%VNORMAL,%P 2:swp_60_0207
;ENDFOLD
;FOLD PTP swp_60_0207 PDAT62 SPOT Gun=2 RETR CLS PGNO1=81 ACTIVE=1 Tool[2]:Gun C2 Base[2]:Accelo;%{PE}%R 8.2.2,%MKUKATPSPOT,%CSPOT,%VPTP,%P 1:PTP, 2:swp_60_0207, 3:, 5:100, 7:PDAT62, 10:2, 12:#FIRST, 14:#CLO, 16:122, 18:1, 20:0, 22:0, 24:1, 25:NORMAL
$BWDSTART=FALSE
PDAT_ACT=PPDAT62
FDAT_ACT=Fswp_60_0207
BAS(#PTP_PARAMS,PPDAT62.VEL)
S_ACT.GUN=2
S_ACT.PAIR=SDEFAULT.PAIR
S_ACT.RETR=#CLO
S_ACT.CLO_TM=1
S_ACT.PGNO1=81
S_ACT.PGNO2=SDEFAULT.PGNO2
S_ACT.PRESS1=SDEFAULT.PRESS1
S_ACT.PRESS2=SDEFAULT.PRESS2
S_READY=FALSE
PTP Xswp_60_0207
USERSPOT(#SPOT, S_ACT)
WAIT FOR S_READY
;ENDFOLD

;FOLD ; swp_60_0209;%{PE}%R 8.2.20,%MKUKATPBASIS,%CCOMMENT,%VNORMAL,%P 2:swp_60_0209
;ENDFOLD
;FOLD PTP swp_60_0209 P_OLP84 SPOT Gun=2 RETR CLS PGNO1=122 ACTIVE=1 Tool[2]:Gun C2 Base[2]:Accelo;%{PE}%R 8.2.2,%MKUKATPSPOT,%CSPOT,%VPTP,%P 1:PTP, 2:swp_60_0209, 3:, 5:100, 7:P_OLP84, 10:2, 12:#FIRST, 14:#CLO, 16:163, 18:1, 20:1, 22:0, 24:1, 25:S_OLP13
$BWDSTART=FALSE
PDAT_ACT=PP_OLP84
FDAT_ACT=Fswp_60_0209
BAS(#PTP_PARAMS,PP_OLP84.VEL)
S_ACT.GUN=2
S_ACT.PAIR=SDEFAULT.PAIR
S_ACT.RETR=#CLO
S_ACT.CLO_TM=1
S_ACT.PGNO1=122
S_ACT.PGNO2=SDEFAULT.PGNO2
S_ACT.PRESS1=SDEFAULT.PRESS1
S_ACT.PRESS2=SDEFAULT.PRESS2
S_READY=FALSE
PTP Xswp_60_0209
USERSPOT(#SPOT, S_ACT)
WAIT FOR S_READY
;ENDFOLD

;FOLD ; swp_60_0211;%{PE}%R 8.2.20,%MKUKATPBASIS,%CCOMMENT,%VNORMAL,%P 2:swp_60_0211
;ENDFOLD
;FOLD PTP swp_60_0211 PDAT63 SPOT Gun=2 RETR OPN PGNO1=80 ACTIVE=1 Tool[2]:Gun C2 Base[2]:Accelo;%{PE}%R 8.2.2,%MKUKATPSPOT,%CSPOT,%VPTP,%P 1:PTP, 2:swp_60_0211, 3:, 5:100, 7:PDAT63, 10:2, 12:#FIRST, 14:#OPN, 16:121, 18:1, 20:0, 22:0, 24:1, 25:NORMAL
$BWDSTART=FALSE
PDAT_ACT=PPDAT63
FDAT_ACT=Fswp_60_0211
BAS(#PTP_PARAMS,PPDAT63.VEL)
S_ACT.GUN=2
S_ACT.PAIR=SDEFAULT.PAIR
S_ACT.RETR=#OPN
S_ACT.CLO_TM=1
S_ACT.PGNO1=80
S_ACT.PGNO2=SDEFAULT.PGNO2
S_ACT.PRESS1=SDEFAULT.PRESS1
S_ACT.PRESS2=SDEFAULT.PRESS2
S_READY=FALSE
PTP Xswp_60_0211
USERSPOT(#SPOT, S_ACT)
WAIT FOR S_READY
;ENDFOLD

;FOLD PTP lx796 CONT Vel=100 % P_OLP51 Tool[2]:Gun C2 Base[2]:Accelo;%{PE}%R 8.2.20,%MKUKATPBASIS,%CMOVE,%VPTP,%P 1:PTP, 2:lx796, 3:C_DIS, 5:100, 7:P_OLP51
$BWDSTART=FALSE
PDAT_ACT=PP_OLP51
FDAT_ACT=Flx796
BAS(#PTP_PARAMS,100)
PTP Xlx796 C_DIS
;ENDFOLD

;FOLD ; swp_60_0205;%{PE}%R 5.4.33,%MKUKATPBASIS,%CCOMMENT,%VNORMAL,%P 2:swp_60_0205
;ENDFOLD
;FOLD PTP swp_60_0205 P_OLP52 SPOT Gun=2 RETR OPN PGNO1=121 ACTIVE=1 Tool[2]:Gun C2 Base[2]:Accelo;%{PE}%R 8.2.2,%MKUKATPSPOT,%CSPOT,%VPTP,%P 1:PTP, 2:swp_60_0205, 3:, 5:100, 7:P_OLP52, 10:2, 12:#FIRST, 14:#OPN, 16:162, 18:1, 20:1, 22:0, 24:1, 25:S_OLP12
$BWDSTART=FALSE
PDAT_ACT=PP_OLP52
FDAT_ACT=Fswp_60_0205
BAS(#PTP_PARAMS,PP_OLP52.VEL)
S_ACT.GUN=2
S_ACT.PAIR=SDEFAULT.PAIR
S_ACT.RETR=#OPN
S_ACT.CLO_TM=1
S_ACT.PGNO1=121
S_ACT.PGNO2=SDEFAULT.PGNO2
S_ACT.PRESS1=SDEFAULT.PRESS1
S_ACT.PRESS2=SDEFAULT.PRESS2
S_READY=FALSE
PTP Xswp_60_0205
USERSPOT(#SPOT, S_ACT)
WAIT FOR S_READY
;ENDFOLD

;FOLD PTP P51 CONT Vel=100 % PDAT65 Tool[2]:Gun C2 Base[2]:Accelo;%{PE}%R 8.2.20,%MKUKATPBASIS,%CMOVE,%VPTP,%P 1:PTP, 2:P51, 3:C_DIS, 5:100, 7:PDAT65
$BWDSTART=FALSE
PDAT_ACT=PPDAT65
FDAT_ACT=FP51
BAS(#PTP_PARAMS,100)
PTP XP51 C_DIS
;ENDFOLD

;FOLD ; swp_60_0203;%{PE}%R 8.2.20,%MKUKATPBASIS,%CCOMMENT,%VNORMAL,%P 2:swp_60_0203
;ENDFOLD
;FOLD PTP swp_60_0203 PDAT76 SPOT Gun=2 RETR CLS PGNO1=82 ACTIVE=1 Tool[2]:Gun C2 Base[2]:Accelo;%{PE}%R 8.2.2,%MKUKATPSPOT,%CSPOT,%VPTP,%P 1:PTP, 2:swp_60_0203, 3:, 5:100, 7:PDAT76, 10:2, 12:#FIRST, 14:#CLO, 16:123, 18:1, 20:0, 22:0, 24:1, 25:NORMAL
$BWDSTART=FALSE
PDAT_ACT=PPDAT76
FDAT_ACT=Fswp_60_0203
BAS(#PTP_PARAMS,PPDAT76.VEL)
S_ACT.GUN=2
S_ACT.PAIR=SDEFAULT.PAIR
S_ACT.RETR=#CLO
S_ACT.CLO_TM=1
S_ACT.PGNO1=82
S_ACT.PGNO2=SDEFAULT.PGNO2
S_ACT.PRESS1=SDEFAULT.PRESS1
S_ACT.PRESS2=SDEFAULT.PRESS2
S_READY=FALSE
PTP Xswp_60_0203
USERSPOT(#SPOT, S_ACT)
WAIT FOR S_READY
;ENDFOLD

;FOLD ; swp_60_0201;%{PE}%R 8.2.20,%MKUKATPBASIS,%CCOMMENT,%VNORMAL,%P 2:swp_60_0201
;ENDFOLD
;FOLD PTP swp_60_0201 P_OLP91 SPOT Gun=2 RETR OPN PGNO1=125 ACTIVE=1 Tool[2]:Gun C2 Base[2]:Accelo;%{PE}%R 8.2.2,%MKUKATPSPOT,%CSPOT,%VPTP,%P 1:PTP, 2:swp_60_0201, 3:, 5:100, 7:P_OLP91, 10:2, 12:#FIRST, 14:#OPN, 16:166, 18:1, 20:1, 22:0, 24:1, 25:S_OLP16
$BWDSTART=FALSE
PDAT_ACT=PP_OLP91
FDAT_ACT=Fswp_60_0201
BAS(#PTP_PARAMS,PP_OLP91.VEL)
S_ACT.GUN=2
S_ACT.PAIR=SDEFAULT.PAIR
S_ACT.RETR=#OPN
S_ACT.CLO_TM=1
S_ACT.PGNO1=125
S_ACT.PGNO2=SDEFAULT.PGNO2
S_ACT.PRESS1=SDEFAULT.PRESS1
S_ACT.PRESS2=SDEFAULT.PRESS2
S_READY=FALSE
PTP Xswp_60_0201
USERSPOT(#SPOT, S_ACT)
WAIT FOR S_READY
;ENDFOLD

;FOLD PTP P63 CONT Vel=100 % PDAT77 Tool[2]:Gun C2 Base[2]:Accelo;%{PE}%R 8.2.20,%MKUKATPBASIS,%CMOVE,%VPTP,%P 1:PTP, 2:P63, 3:C_DIS, 5:100, 7:PDAT77
$BWDSTART=FALSE
PDAT_ACT=PPDAT77
FDAT_ACT=FP63
BAS(#PTP_PARAMS,100)
PTP XP63 C_DIS
;ENDFOLD
;FOLD PTP P64 CONT Vel=100 % PDAT78 Tool[2]:Gun C2 Base[2]:Accelo;%{PE}%R 8.2.20,%MKUKATPBASIS,%CMOVE,%VPTP,%P 1:PTP, 2:P64, 3:C_DIS, 5:100, 7:PDAT78
$BWDSTART=FALSE
PDAT_ACT=PPDAT78
FDAT_ACT=FP64
BAS(#PTP_PARAMS,100)
PTP XP64 C_DIS
;ENDFOLD
;FOLD PTP P53 CONT Vel=100 % PDAT67 Tool[2]:Gun C2 Base[2]:Accelo;%{PE}%R 8.2.20,%MKUKATPBASIS,%CMOVE,%VPTP,%P 1:PTP, 2:P53, 3:C_DIS, 5:100, 7:PDAT67
$BWDSTART=FALSE
PDAT_ACT=PPDAT67
FDAT_ACT=FP53
BAS(#PTP_PARAMS,100)
PTP XP53 C_DIS
;ENDFOLD
;FOLD PTP P0 CONT Vel=100 % PDAT0 Tool[2]:Gun C2 Base[2]:Accelo;%{PE}%R 8.2.20,%MKUKATPBASIS,%CMOVE,%VPTP,%P 1:PTP, 2:P0, 3:C_DIS, 5:100, 7:PDAT0
$BWDSTART=FALSE
PDAT_ACT=PPDAT0
FDAT_ACT=FP0
BAS(#PTP_PARAMS,100)
PTP XP0 C_DIS
;ENDFOLD
;FOLD PTP P55 CONT Vel=100 % PDAT69 Tool[2]:Gun C2 Base[2]:Accelo;%{PE}%R 8.2.20,%MKUKATPBASIS,%CMOVE,%VPTP,%P 1:PTP, 2:P55, 3:C_DIS, 5:100, 7:PDAT69
$BWDSTART=FALSE
PDAT_ACT=PPDAT69
FDAT_ACT=FP55
BAS(#PTP_PARAMS,100)
PTP XP55 C_DIS
;ENDFOLD
;FOLD PTP P56 CONT Vel=100 % PDAT70 Tool[2]:Gun C2 Base[2]:Accelo;%{PE}%R 8.2.20,%MKUKATPBASIS,%CMOVE,%VPTP,%P 1:PTP, 2:P56, 3:C_DIS, 5:100, 7:PDAT70
$BWDSTART=FALSE
PDAT_ACT=PPDAT70
FDAT_ACT=FP56
BAS(#PTP_PARAMS,100)
PTP XP56 C_DIS
;ENDFOLD
;FOLD PTP P57 CONT Vel=80 % PDAT71 Tool[2]:Gun C2 Base[2]:Accelo;%{PE}%R 8.2.20,%MKUKATPBASIS,%CMOVE,%VPTP,%P 1:PTP, 2:P57, 3:C_DIS, 5:80, 7:PDAT71
$BWDSTART=FALSE
PDAT_ACT=PPDAT71
FDAT_ACT=FP57
BAS(#PTP_PARAMS,80)
PTP XP57 C_DIS
;ENDFOLD

;FOLD ; swp_60_0217;%{PE}%R 8.2.20,%MKUKATPBASIS,%CCOMMENT,%VNORMAL,%P 2:swp_60_0217
;ENDFOLD
;FOLD PTP swp_60_0217 P_OLP86 SPOT Gun=2 RETR CLS PGNO1=123 ACTIVE=1 Tool[2]:Gun C2 Base[2]:Accelo;%{PE}%R 8.2.2,%MKUKATPSPOT,%CSPOT,%VPTP,%P 1:PTP, 2:swp_60_0217, 3:, 5:100, 7:P_OLP86, 10:2, 12:#FIRST, 14:#CLO, 16:164, 18:1, 20:1, 22:0, 24:1, 25:S_OLP14
$BWDSTART=FALSE
PDAT_ACT=PP_OLP86
FDAT_ACT=Fswp_60_0217
BAS(#PTP_PARAMS,PP_OLP86.VEL)
S_ACT.GUN=2
S_ACT.PAIR=SDEFAULT.PAIR
S_ACT.RETR=#CLO
S_ACT.CLO_TM=1
S_ACT.PGNO1=123
S_ACT.PGNO2=SDEFAULT.PGNO2
S_ACT.PRESS1=SDEFAULT.PRESS1
S_ACT.PRESS2=SDEFAULT.PRESS2
S_READY=FALSE
PTP Xswp_60_0217
USERSPOT(#SPOT, S_ACT)
WAIT FOR S_READY
;ENDFOLD

;FOLD ; swp_60_0219;%{PE}%R 8.2.20,%MKUKATPBASIS,%CCOMMENT,%VNORMAL,%P 2:swp_60_0219
;ENDFOLD
;FOLD PTP swp_60_0219 P_OLP87 SPOT Gun=2 RETR OPN PGNO1=124 ACTIVE=1 Tool[2]:Gun C2 Base[2]:Accelo;%{PE}%R 8.2.2,%MKUKATPSPOT,%CSPOT,%VPTP,%P 1:PTP, 2:swp_60_0219, 3:, 5:100, 7:P_OLP87, 10:2, 12:#FIRST, 14:#OPN, 16:165, 18:1, 20:1, 22:0, 24:1, 25:S_OLP15
$BWDSTART=FALSE
PDAT_ACT=PP_OLP87
FDAT_ACT=Fswp_60_0219
BAS(#PTP_PARAMS,PP_OLP87.VEL)
S_ACT.GUN=2
S_ACT.PAIR=SDEFAULT.PAIR
S_ACT.RETR=#OPN
S_ACT.CLO_TM=1
S_ACT.PGNO1=124
S_ACT.PGNO2=SDEFAULT.PGNO2
S_ACT.PRESS1=SDEFAULT.PRESS1
S_ACT.PRESS2=SDEFAULT.PRESS2
S_READY=FALSE
PTP Xswp_60_0219
USERSPOT(#SPOT, S_ACT)
WAIT FOR S_READY
;ENDFOLD

;FOLD PTP lx788 CONT Vel=100 % P_OLP88 Tool[2]:Gun C2 Base[2]:Accelo;%{PE}%R 8.2.20,%MKUKATPBASIS,%CMOVE,%VPTP,%P 1:PTP, 2:lx788, 3:C_DIS, 5:100, 7:P_OLP88
$BWDSTART=FALSE
PDAT_ACT=PP_OLP88
FDAT_ACT=Flx788
BAS(#PTP_PARAMS,100)
PTP Xlx788 C_DIS
;ENDFOLD
;FOLD PTP lx831 CONT Vel=100 % P_OLP89 Tool[2]:Gun C2 Base[2]:Accelo;%{PE}%R 8.2.20,%MKUKATPBASIS,%CMOVE,%VPTP,%P 1:PTP, 2:lx831, 3:C_DIS, 5:100, 7:P_OLP89
$BWDSTART=FALSE
PDAT_ACT=PP_OLP89
FDAT_ACT=Flx831
BAS(#PTP_PARAMS,100)
PTP Xlx831 C_DIS
;ENDFOLD
;FOLD PTP P59 CONT Vel=100 % PDAT73 Tool[2]:Gun C2 Base[2]:Accelo;%{PE}%R 8.2.20,%MKUKATPBASIS,%CMOVE,%VPTP,%P 1:PTP, 2:P59, 3:C_DIS, 5:100, 7:PDAT73
$BWDSTART=FALSE
PDAT_ACT=PPDAT73
FDAT_ACT=FP59
BAS(#PTP_PARAMS,100)
PTP XP59 C_DIS
;ENDFOLD
;FOLD PTP lx780 Vel=100 % P_OLP71 Tool[2]:Gun C2 Base[2]:Accelo;%{PE}%R 8.2.20,%MKUKATPBASIS,%CMOVE,%VPTP,%P 1:PTP, 2:lx780, 3:, 5:100, 7:P_OLP71
$BWDSTART=FALSE
PDAT_ACT=PP_OLP71
FDAT_ACT=Flx780
BAS(#PTP_PARAMS,100)
PTP Xlx780
;ENDFOLD

;FOLD Collision.Monitoring_AREA_3_Off . ;%{PE}%MKUKATPUSER
COLLSTOP( 9, 2+0 )
;ENDFOLD
end_weld_geo ( )
;FOLD OUT 3348 'Fora area GEOBOX' State=TRUE ;%{PE}%R 8.2.20,%MKUKATPBASIS,%COUT,%VOUTX,%P 2:3348, 3:Fora area GEOBOX, 5:TRUE, 6:
$OUT[3348]=TRUE
;ENDFOLD

;FOLD PTP lx767 CONT Vel=100 % P_OLP81 Tool[2]:Gun C2 Base[2]:Accelo;%{PE}%R 8.2.20,%MKUKATPBASIS,%CMOVE,%VPTP,%P 1:PTP, 2:lx767, 3:C_DIS, 5:100, 7:P_OLP81
$BWDSTART=FALSE
PDAT_ACT=PP_OLP81
FDAT_ACT=Flx767
BAS(#PTP_PARAMS,100)
PTP Xlx767 C_DIS
;ENDFOLD
;FOLD PTP P47 CONT Vel=100 % PDAT51 Tool[2]:Gun C2 Base[2]:Accelo;%{PE}%R 8.2.20,%MKUKATPBASIS,%CMOVE,%VPTP,%P 1:PTP, 2:P47, 3:C_DIS, 5:100, 7:PDAT51
$BWDSTART=FALSE
PDAT_ACT=PPDAT51
FDAT_ACT=FP47
BAS(#PTP_PARAMS,100)
PTP XP47 C_DIS
;ENDFOLD

IF (NOT(GHOST())) THEN
if FraesAnf (2) then
  f_fraes2 ()
endif
ENDIF


END

--- ps_ltc_geo_c2_bolha.dat ---
&ACCESS RVO1
&REL 3
&COMMENT GUN C2 geom Accelo
&PARAM DISKPATH = KRC:\R1\Program
DEFDAT  ps_ltc_geo_c2_bolha
;FOLD EXTERNAL DECLARATIONS;%{PE}%MKUKATPBASIS,%CEXT,%VCOMMON,%P
;FOLD GRIPPERTECH EXT
EXT  H50 (INT  :IN,INT  :IN,INT  :IN,GRP_TYP  :IN )
;ENDFOLD (GRIPPERTECH EXT)
;FOLD SPOTTECH EXT
EXT  USERSPOT (S_COMMAND  :IN,SPOT_TYPE  :IN )
;ENDFOLD (SPOTTECH EXT)
;FOLD BASISTECH EXT;%{PE}%MKUKATPBASIS,%CEXT,%VEXT,%P
EXT  BAS (BAS_COMMAND  :IN,REAL  :IN )
DECL INT SUCCESS
;ENDFOLD (BASISTECH EXT)
;FOLD USER EXT;%{E}%MKUKATPUSER,%CEXT,%VEXT,%P
;Make your modifications here

;ENDFOLD (USER EXT)
;ENDFOLD (EXTERNAL DECLARATIONS)
;# ============ START PATH : swp_p13050r3_ltc_geo_c2 =============
DECL FDAT Flx828={TOOL_NO 2,BASE_NO 2,IPO_FRAME #BASE,POINT2[] " "}
DECL PDAT PP_OLP7={VEL 100.0,ACC 100.0,APO_DIST 30.0,APO_MODE #CDIS}
DECL E6POS Xlx828={X 1313.89404,Y -1331.46704,Z 523.221985,A -13.1561899,B 25.8715191,C 86.3671722,S 2,T 11,E1 5636.96094,E2 0.0,E3 0.0,E4 0.0,E5 0.0,E6 0.0}
DECL FDAT Flx827={TOOL_NO 2,BASE_NO 2,IPO_FRAME #BASE,POINT2[] " "}
DECL PDAT PP_OLP8={VEL 100.0,ACC 100.0,APO_DIST 30.0,APO_MODE #CDIS}
DECL E6POS Xlx827={X 1268.92896,Y -1028.29199,Z 484.852692,A 0.744642675,B 44.8028793,C 92.9150925,S 2,T 11,E1 5636.54883,E2 0.0,E3 0.0,E4 0.0,E5 0.0,E6 0.0}
DECL FDAT Flx826={TOOL_NO 2,BASE_NO 2,IPO_FRAME #BASE,POINT2[] " "}
DECL PDAT PP_OLP9={VEL 100.0,ACC 100.0,APO_DIST 100.0,APO_MODE #CDIS}
DECL E6POS Xlx826={X 1247.14197,Y -839.330017,Z 487.233398,A 0.873326421,B 46.5667191,C 93.0090027,S 2,T 11,E1 5636.54297,E2 0.0,E3 0.0,E4 0.0,E5 0.0,E6 0.0}
DECL FDAT Fswp_60_0399={TOOL_NO 2,BASE_NO 2,IPO_FRAME #BASE,POINT2[] " "}
DECL PDAT PP_OLP10={VEL 100.0,ACC 100.0,APO_DIST 0.0}
DECL SPOT_TYPE SS_OLP1={GUN 1,PAIR #FIRST,RETR #OPN,CLO_TM 0,PGNO1 1,PRESS1 1.0,PGNO2 0,PRESS2 0.0}
DECL E6POS Xswp_60_0399={X 1474.20605,Y -844.474304,Z 742.124817,A 0.666326225,B -12.8174696,C 91.9340897,S 2,T 11,E1 5636.55811,E2 0.0,E3 0.0,E4 0.0,E5 0.0,E6 0.0}
DECL FDAT Fswp_60_0395={TOOL_NO 2,BASE_NO 2,IPO_FRAME #BASE,POINT2[] " "}
DECL PDAT PP_OLP12={VEL 100.0,ACC 100.0,APO_DIST 0.0}
DECL SPOT_TYPE SS_OLP2={GUN 1,PAIR #FIRST,RETR #OPN,CLO_TM 0,PGNO1 1,PRESS1 1.0,PGNO2 0,PRESS2 0.0}
DECL E6POS Xswp_60_0395={X 1445.07202,Y -842.604614,Z 672.663025,A 1.23996997,B -7.01102686,C 91.9965591,S 2,T 11,E1 5636.50488,E2 0.0,E3 0.0,E4 0.0,E5 0.0,E6 0.0}
DECL FDAT Flx824={TOOL_NO 2,BASE_NO 2,IPO_FRAME #BASE,POINT2[] " "}
DECL PDAT PP_OLP13={VEL 100.0,ACC 100.0,APO_DIST 100.0,APO_MODE #CDIS}
DECL E6POS Xlx824={X 1443.104,Y -839.287109,Z 639.178406,A 2.08833504,B 1.78453195,C 92.0118713,S 2,T 11,E1 5636.50488,E2 0.0,E3 0.0,E4 0.0,E5 0.0,E6 0.0}
DECL FDAT Fswp_60_0393={TOOL_NO 2,BASE_NO 2,IPO_FRAME #BASE,POINT2[] " "}
DECL PDAT PP_OLP14={VEL 100.0,ACC 100.0,APO_DIST 0.0}
DECL SPOT_TYPE SS_OLP3={GUN 1,PAIR #FIRST,RETR #OPN,CLO_TM 0,PGNO1 1,PRESS1 1.0,PGNO2 0,PRESS2 0.0}
DECL E6POS Xswp_60_0393={X 1465.23303,Y -844.253113,Z 638.954773,A -0.0227528401,B 3.38127303,C 92.2101974,S 2,T 11,E1 5636.49512,E2 0.0,E3 0.0,E4 0.0,E5 0.0,E6 0.0}
DECL FDAT Flx823={TOOL_NO 2,BASE_NO 2,IPO_FRAME #BASE,POINT2[] " "}
DECL PDAT PP_OLP16={VEL 100.0,ACC 100.0,APO_DIST 100.0,APO_MODE #CDIS}
DECL E6POS Xlx823={X 1363.30005,Y -822.437317,Z 549.010315,A 0.472675204,B 20.0343704,C 92.5931931,S 2,T 11,E1 5636.54199,E2 0.0,E3 0.0,E4 0.0,E5 0.0,E6 0.0}
DECL FDAT Flx820={TOOL_NO 2,BASE_NO 2,IPO_FRAME #BASE,POINT2[] " "}
DECL PDAT PP_OLP18={VEL 100.0,ACC 100.0,APO_DIST 100.0,APO_MODE #CDIS}
DECL E6POS Xlx820={X 1251.099,Y -1023.78699,Z 483.461304,A 0.771801889,B 44.3958397,C 93.1082611,S 2,T 11,E1 5636.50977,E2 0.0,E3 0.0,E4 0.0,E5 0.0,E6 0.0}
DECL FDAT Flx819={TOOL_NO 2,BASE_NO 2,IPO_FRAME #BASE,POINT2[] " "}
DECL PDAT PP_OLP19={VEL 100.0,ACC 100.0,APO_DIST 100.0,APO_MODE #CDIS}
DECL E6POS Xlx819={X 1444.45801,Y -1414.67004,Z 462.043915,A -12.3754196,B 44.4594803,C 91.9307175,S 2,T 11,E1 5636.50586,E2 0.0,E3 0.0,E4 0.0,E5 0.0,E6 0.0}
DECL FDAT Fswp_60_0341={TOOL_NO 2,BASE_NO 2,IPO_FRAME #BASE,POINT2[] " "}
DECL PDAT PP_OLP21={VEL 100.0,ACC 100.0,APO_DIST 0.0}
DECL SPOT_TYPE SS_OLP4={GUN 1,PAIR #FIRST,RETR #OPN,CLO_TM 0,PGNO1 1,PRESS1 1.0,PGNO2 0,PRESS2 0.0}
DECL E6POS Xswp_60_0341={X 1400.88696,Y -841.813171,Z 60.6647987,A -3.50004601,B 32.0640984,C 89.0238266,S 2,T 11,E1 5553.2959,E2 0.0,E3 0.0,E4 0.0,E5 0.0,E6 0.0}
DECL FDAT Fswp_60_0333={TOOL_NO 2,BASE_NO 2,IPO_FRAME #BASE,POINT2[] " "}
DECL PDAT PP_OLP22={VEL 100.0,ACC 100.0,APO_DIST 0.0}
DECL SPOT_TYPE SS_OLP5={GUN 1,PAIR #FIRST,RETR #OPN,CLO_TM 0,PGNO1 1,PRESS1 1.0,PGNO2 0,PRESS2 0.0}
DECL E6POS Xswp_60_0333={X 1245.823,Y -840.628174,Z 60.1122894,A -3.49715209,B 31.6406898,C 88.9972,S 2,T 11,E1 5553.13379,E2 0.0,E3 0.0,E4 0.0,E5 0.0,E6 0.0}
DECL FDAT Flx815={TOOL_NO 2,BASE_NO 2,IPO_FRAME #BASE,POINT2[] " "}
DECL PDAT PP_OLP23={VEL 100.0,ACC 100.0,APO_DIST 100.0,APO_MODE #CDIS}
DECL E6POS Xlx815={X 1196.84094,Y -826.712402,Z 159.871796,A -3.81221008,B 31.1064892,C 88.8207474,S 2,T 11,E1 5552.36182,E2 0.0,E3 0.0,E4 0.0,E5 0.0,E6 0.0}
DECL FDAT Flx816={TOOL_NO 2,BASE_NO 2,IPO_FRAME #BASE,POINT2[] " "}
DECL PDAT PP_OLP24={VEL 100.0,ACC 100.0,APO_DIST 30.0,APO_MODE #CDIS}
DECL E6POS Xlx816={X 1198.349,Y -1363.80798,Z 157.276199,A -10.3484898,B 31.0169201,C 86.4901962,S 2,T 11,E1 5539.03516,E2 0.0,E3 0.0,E4 0.0,E5 0.0,E6 0.0}
DECL FDAT Flx814={TOOL_NO 2,BASE_NO 2,IPO_FRAME #BASE,POINT2[] " "}
DECL E6POS Xlx814={X 369.932312,Y -1519.18604,Z -172.970001,A -167.901596,B 57.7843094,C -67.7142334,S 2,T 11,E1 4678.13623,E2 0.0,E3 0.0,E4 0.0,E5 0.0,E6 0.0}
DECL FDAT Flx813={TOOL_NO 2,BASE_NO 2,IPO_FRAME #BASE,POINT2[] " "}
DECL E6POS Xlx813={X 428.942688,Y -806.54657,Z -98.9288864,A 175.669601,B 53.0529213,C -91.0339203,S 2,T 11,E1 4678.10986,E2 0.0,E3 0.0,E4 0.0,E5 0.0,E6 0.0}
DECL FDAT Fswp_60_0255={TOOL_NO 2,BASE_NO 2,IPO_FRAME #BASE,POINT2[] " "}
DECL PDAT PP_OLP30={VEL 100.0,ACC 100.0,APO_DIST 0.0}
DECL SPOT_TYPE SS_OLP6={GUN 1,PAIR #FIRST,RETR #OPN,CLO_TM 0,PGNO1 1,PRESS1 1.0,PGNO2 0,PRESS2 0.0}
DECL E6POS Xswp_60_0255={X 300.463989,Y -853.163086,Z -119.2994,A 175.893997,B 45.7151489,C -93.9277267,S 2,T 11,E1 4678.07178,E2 0.0,E3 0.0,E4 0.0,E5 0.0,E6 0.0}
DECL FDAT Fswp_60_0245={TOOL_NO 2,BASE_NO 2,IPO_FRAME #BASE,POINT2[] " "}
DECL PDAT PP_OLP31={VEL 100.0,ACC 100.0,APO_DIST 0.0}
DECL SPOT_TYPE SS_OLP7={GUN 1,PAIR #FIRST,RETR #OPN,CLO_TM 0,PGNO1 1,PRESS1 1.0,PGNO2 0,PRESS2 0.0}
DECL E6POS Xswp_60_0245={X 236.971893,Y -854.070374,Z -10.8238602,A -179.4767,B 23.06007,C -91.1865311,S 2,T 11,E1 4684.35791,E2 0.0,E3 0.0,E4 0.0,E5 0.0,E6 0.0}
DECL FDAT Fswp_60_0235={TOOL_NO 2,BASE_NO 2,IPO_FRAME #BASE,POINT2[] " "}
DECL PDAT PP_OLP33={VEL 100.0,ACC 100.0,APO_DIST 0.0}
DECL SPOT_TYPE SS_OLP8={GUN 1,PAIR #FIRST,RETR #OPN,CLO_TM 0,PGNO1 1,PRESS1 1.0,PGNO2 0,PRESS2 0.0}
DECL E6POS Xswp_60_0235={X 258.574402,Y -852.900208,Z 151.175507,A -179.494904,B -23.2381096,C -89.6756897,S 2,T 11,E1 4681.46387,E2 0.0,E3 0.0,E4 0.0,E5 0.0,E6 0.0}
DECL FDAT Flx798={TOOL_NO 2,BASE_NO 2,IPO_FRAME #BASE,POINT2[] " "}
DECL PDAT PP_OLP34={VEL 100.0,ACC 100.0,APO_DIST 100.0,APO_MODE #CDIS}
DECL E6POS Xlx798={X 268.457794,Y -793.195618,Z 67.879303,A -179.860504,B 7.61739111,C -89.3985977,S 2,T 11,E1 4683.8208,E2 0.0,E3 0.0,E4 0.0,E5 0.0,E6 0.0}
DECL FDAT Flx799={TOOL_NO 2,BASE_NO 2,IPO_FRAME #BASE,POINT2[] " "}
DECL PDAT PP_OLP35={VEL 100.0,ACC 100.0,APO_DIST 100.0,APO_MODE #CDIS}
DECL E6POS Xlx799={X 345.372589,Y -812.418274,Z -84.5929871,A 176.158905,B 42.65382,C -93.2365875,S 2,T 11,E1 4677.79199,E2 0.0,E3 0.0,E4 0.0,E5 0.0,E6 0.0}
DECL FDAT Flx800={TOOL_NO 2,BASE_NO 2,IPO_FRAME #BASE,POINT2[] " "}
DECL E6POS Xlx800={X 428.928711,Y -806.551819,Z -98.9253006,A 175.669693,B 53.0524902,C -91.0339737,S 2,T 11,E1 4686.33398,E2 0.0,E3 0.0,E4 0.0,E5 0.0,E6 0.0}
DECL FDAT Flx802={TOOL_NO 2,BASE_NO 2,IPO_FRAME #BASE,POINT2[] " "}
DECL PDAT PP_OLP37={VEL 100.0,ACC 100.0,APO_DIST 100.0,APO_MODE #CDIS}
DECL E6POS Xlx802={X 410.083588,Y -1114.28699,Z -102.263397,A 175.624405,B 54.5072289,C -91.0710373,S 2,T 11,E1 4684.38477,E2 0.0,E3 0.0,E4 0.0,E5 0.0,E6 0.0}
DECL FDAT Flx801={TOOL_NO 2,BASE_NO 2,IPO_FRAME #BASE,POINT2[] " "}
DECL PDAT PP_OLP38={VEL 100.0,ACC 100.0,APO_DIST 10.0,APO_MODE #CDIS}
DECL E6POS Xlx801={X 350.765411,Y -1468.63098,Z -154.114105,A -172.531601,B 56.018959,C -75.8321533,S 2,T 11,E1 4678.13477,E2 0.0,E3 0.0,E4 0.0,E5 0.0,E6 0.0}
DECL FDAT Flx804={TOOL_NO 2,BASE_NO 2,IPO_FRAME #BASE,POINT2[] " "}
DECL E6POS Xlx804={X 395.674713,Y -813.304382,Z 335.053406,A -179.504196,B 41.2089806,C -87.9716721,S 2,T 11,E1 4687.36084,E2 0.0,E3 0.0,E4 0.0,E5 0.0,E6 0.0}
DECL FDAT Flx803={TOOL_NO 2,BASE_NO 2,IPO_FRAME #BASE,POINT2[] " "}
DECL PDAT PP_OLP45={VEL 100.0,ACC 100.0,APO_DIST 100.0,APO_MODE #CDIS}
DECL E6POS Xlx803={X 236.066498,Y -818.786377,Z 292.583099,A -179.961105,B 26.3373394,C -89.4697876,S 2,T 11,E1 4682.87988,E2 0.0,E3 0.0,E4 0.0,E5 0.0,E6 0.0}
DECL FDAT Fswp_60_0229={TOOL_NO 2,BASE_NO 2,IPO_FRAME #BASE,POINT2[] " ",TQ_STATE FALSE}
DECL PDAT PP_OLP46={VEL 100.0,ACC 100.0,APO_DIST 0.0}
DECL SPOT_TYPE SS_OLP9={GUN 1,PAIR #FIRST,RETR #OPN,CLO_TM 0,PGNO1 1,PRESS1 1.0,PGNO2 0,PRESS2 0.0}
DECL E6POS Xswp_60_0229={X 213.870193,Y -866.033508,Z 246.082993,A -179.964996,B 26.52174,C -89.4645767,S 2,T 11,E1 4685.67676,E2 0.0,E3 0.0,E4 0.0,E5 0.0,E6 0.0}
DECL FDAT Fswp_60_0225={TOOL_NO 2,BASE_NO 2,IPO_FRAME #BASE,POINT2[] " "}
DECL PDAT PP_OLP47={VEL 100.0,ACC 100.0,APO_DIST 0.0}
DECL SPOT_TYPE SS_OLP10={GUN 1,PAIR #FIRST,RETR #OPN,CLO_TM 0,PGNO1 1,PRESS1 1.0,PGNO2 0,PRESS2 0.0}
DECL E6POS Xswp_60_0225={X 207.132599,Y -867.208618,Z 281.93811,A -178.352097,B 25.9885197,C -88.7658081,S 2,T 11,E1 4685.66797,E2 0.0,E3 0.0,E4 0.0,E5 0.0,E6 0.0}
DECL FDAT Fswp_60_0221={TOOL_NO 2,BASE_NO 2,IPO_FRAME #BASE,POINT2[] " "}
DECL PDAT PP_OLP49={VEL 100.0,ACC 100.0,APO_DIST 0.0}
DECL SPOT_TYPE SS_OLP11={GUN 1,PAIR #FIRST,RETR #OPN,CLO_TM 0,PGNO1 1,PRESS1 1.0,PGNO2 0,PRESS2 0.0}
DECL E6POS Xswp_60_0221={X 171.744797,Y -866.035828,Z 326.67749,A -177.524902,B 4.52732706,C -90.1039963,S 2,T 11,E1 4681.50586,E2 0.0,E3 0.0,E4 0.0,E5 0.0,E6 0.0}
DECL FDAT Flx795={TOOL_NO 2,BASE_NO 2,IPO_FRAME #BASE,POINT2[] " "}
DECL PDAT PP_OLP50={VEL 100.0,ACC 100.0,APO_DIST 100.0,APO_MODE #CDIS}
DECL E6POS Xlx795={X 226.200195,Y -837.525085,Z 348.480286,A -178.942001,B 2.25270796,C -89.7577896,S 2,T 11,E1 4678.92383,E2 0.0,E3 0.0,E4 0.0,E5 0.0,E6 0.0}
DECL FDAT Flx796={TOOL_NO 2,BASE_NO 2,IPO_FRAME #BASE,POINT2[] " "}
DECL PDAT PP_OLP51={VEL 100.0,ACC 100.0,APO_DIST 100.0,APO_MODE #CDIS}
DECL E6POS Xlx796={X 263.717407,Y -815.125122,Z 435.898987,A -178.984207,B 0.893851578,C -89.7701492,S 2,T 11,E1 4682.00098,E2 0.0,E3 0.0,E4 0.0,E5 0.0,E6 0.0}
DECL FDAT Fswp_60_0205={TOOL_NO 2,BASE_NO 2,IPO_FRAME #BASE,POINT2[] " "}
DECL PDAT PP_OLP52={VEL 100.0,ACC 100.0,APO_DIST 0.0}
DECL SPOT_TYPE SS_OLP12={GUN 1,PAIR #FIRST,RETR #OPN,CLO_TM 0,PGNO1 1,PRESS1 1.0,PGNO2 0,PRESS2 0.0}
DECL E6POS Xswp_60_0205={X 265.348785,Y -866.557007,Z 493.816589,A -178.943497,B 1.47540104,C -89.7626266,S 2,T 11,E1 4677.98193,E2 0.0,E3 0.0,E4 0.0,E5 0.0,E6 0.0}
DECL FDAT Fswp_60_0209={TOOL_NO 2,BASE_NO 2,IPO_FRAME #BASE,POINT2[] " "}
DECL SPOT_TYPE SS_OLP13={GUN 1,PAIR #FIRST,RETR #OPN,CLO_TM 0,PGNO1 1,PRESS1 1.0,PGNO2 0,PRESS2 0.0}
DECL E6POS Xswp_60_0209={X 198.481094,Y -864.911804,Z 450.41629,A -179.031204,B -7.38108301,C -89.7767487,S 2,T 11,E1 4674.09619,E2 0.0,E3 0.0,E4 0.0,E5 0.0,E6 0.0}
DECL FDAT Fswp_60_0217={TOOL_NO 2,BASE_NO 2,IPO_FRAME #BASE,POINT2[] " "}
DECL SPOT_TYPE SS_OLP14={GUN 1,PAIR #FIRST,RETR #OPN,CLO_TM 0,PGNO1 1,PRESS1 1.0,PGNO2 0,PRESS2 0.0}
DECL E6POS Xswp_60_0217={X 129.435394,Y -861.487915,Z 279.004608,A 17.8512707,B -39.6672592,C 83.1958389,S 2,T 11,E1 4906.23389,E2 0.0,E3 0.0,E4 0.0,E5 0.0,E6 0.0}
DECL FDAT Fswp_60_0219={TOOL_NO 2,BASE_NO 2,IPO_FRAME #BASE,POINT2[] " "}
DECL SPOT_TYPE SS_OLP15={GUN 1,PAIR #FIRST,RETR #OPN,CLO_TM 0,PGNO1 1,PRESS1 1.0,PGNO2 0,PRESS2 0.0}
DECL E6POS Xswp_60_0219={X 132.783798,Y -863.262512,Z 297.808594,A 16.7955704,B -40.7878494,C 86.3009567,S 2,T 11,E1 4905.89502,E2 0.0,E3 0.0,E4 0.0,E5 0.0,E6 0.0}
DECL FDAT Flx780={TOOL_NO 2,BASE_NO 2,IPO_FRAME #BASE,POINT2[] " "}
DECL PDAT PP_OLP71={VEL 100.0,ACC 100.0,APO_DIST 25.0,APO_MODE #CDIS}
DECL E6POS Xlx780={X -536.1073,Y -3036.90088,Z -433.383789,A -103.127502,B 3.39632702,C 10.3325796,S 2,T 11,E1 3967.95703,E2 0.0,E3 0.0,E4 0.0,E5 0.0,E6 0.0}
DECL FDAT Fswp_60_0201={TOOL_NO 2,BASE_NO 2,IPO_FRAME #BASE,POINT2[] " "}
DECL SPOT_TYPE SS_OLP16={GUN 1,PAIR #FIRST,RETR #OPN,CLO_TM 0,PGNO1 1,PRESS1 1.0,PGNO2 0,PRESS2 0.0}
DECL E6POS Xswp_60_0201={X 229.770004,Y -890.145325,Z 555.893982,A -179.049301,B -22.7869892,C -89.742157,S 2,T 11,E1 4680.5332,E2 0.0,E3 0.0,E4 0.0,E5 0.0,E6 0.0}
DECL FDAT Flx767={TOOL_NO 2,BASE_NO 2,IPO_FRAME #BASE,POINT2[] " "}
DECL PDAT PP_OLP81={VEL 100.0,ACC 100.0,APO_DIST 30.0,APO_MODE #CDIS}
DECL E6POS Xlx767={X -4198.59521,Y -2862.68604,Z -364.78479,A 103.820503,B 2.44905901,C -6.20870399,S 2,T 43,E1 1408.61401,E2 0.0,E3 0.0,E4 0.0,E5 0.0,E6 0.0}
DECL BASIS_SUGG_T LAST_BASIS={POINT1[] "PS01010001              ",POINT2[] "PS01010001              ",CP_PARAMS[] "CPDAT0                  ",PTP_PARAMS[] "PDAT0                   ",CONT[] "                        ",CP_VEL[] "2.0                     ",PTP_VEL[] "100                     ",SPL_NAME[] "S0                      "}
DECL E6POS XP2={X -483.254089,Y -2982.05591,Z -402.20639,A -107.179497,B 0.544633925,C 4.32910204,S 2,T 3,E1 4351.56006,E2 0.0,E3 0.0,E4 0.0,E5 0.0,E6 0.0}
DECL FDAT FP2={TOOL_NO 2,BASE_NO 2,IPO_FRAME #BASE,POINT2[] " ",TQ_STATE FALSE}
DECL PDAT PPDAT2={VEL 100.0,ACC 100.0,APO_DIST 30.0,APO_MODE #CDIS}
DECL SPOT_SUGG_T LAST_SPOT={GUN[] "2                       ",RETR_CMD[] "#OPN                    ",CHOISE[] "#FIRST                  ",CLO_TM[] "1                       ",PGNO1[] "252                     ",PRESS1[] "0                       ",PGNO2[] "1                       ",PRESS2[] "0                       ",SPOT_PARAMS[] "NORMAL                  "}
DECL E6POS XP6={X 1279.60999,Y -1373.32605,Z 198.834396,A -9.93967724,B 7.73596001,C 90.3461227,S 2,T 11,E1 5553.88281,E2 0.0,E3 0.0,E4 0.0,E5 0.0,E6 0.0}
DECL FDAT FP6={TOOL_NO 2,BASE_NO 2,IPO_FRAME #BASE,POINT2[] " ",TQ_STATE FALSE}
DECL PDAT PPDAT6={VEL 100.0,ACC 100.0,APO_DIST 30.0,APO_MODE #CDIS}
DECL E6POS XP7={X 1202.75,Y -808.4328,Z 199.5867,A -5.53556919,B 7.68426991,C 92.4831314,S 2,T 11,E1 5553.88184,E2 0.0,E3 0.0,E4 0.0,E5 0.0,E6 0.0}
DECL FDAT FP7={TOOL_NO 2,BASE_NO 2,IPO_FRAME #BASE,POINT2[] " ",TQ_STATE FALSE}
DECL PDAT PPDAT7={VEL 100.0,ACC 100.0,APO_DIST 100.0}
DECL E6POS XP11={X 262.014008,Y -846.799622,Z 144.059601,A -179.474792,B -23.1920395,C -89.2290115,S 2,T 11,E1 4682.82422,E2 0.0,E3 0.0,E4 0.0,E5 0.0,E6 0.0}
DECL FDAT FP11={TOOL_NO 2,BASE_NO 2,IPO_FRAME #BASE,POINT2[] " ",TQ_STATE FALSE}
DECL PDAT PPDAT11={VEL 100.0,ACC 100.0,APO_DIST 10.0,APO_MODE #CDIS}
DECL LDAT LCPDAT1={VEL 2.0,ACC 100.0,APO_DIST 2.0,APO_FAC 50.0,AXIS_VEL 100.0,AXIS_ACC 100.0,ORI_TYP #VAR,CIRC_TYP #BASE,JERK_FAC 50.0,GEAR_JERK 50.0,EXAX_IGN 0}
DECL LDAT LCPDAT5={VEL 2.0,ACC 100.0,APO_DIST 20.0,APO_FAC 50.0,AXIS_VEL 100.0,AXIS_ACC 100.0,ORI_TYP #VAR,CIRC_TYP #BASE,JERK_FAC 50.0,GEAR_JERK 50.0,EXAX_IGN 0}
DECL LDAT LCPDAT8={VEL 2.0,ACC 100.0,APO_DIST 2.0,APO_FAC 50.0,AXIS_VEL 100.0,AXIS_ACC 100.0,ORI_TYP #VAR,CIRC_TYP #BASE,JERK_FAC 50.0,GEAR_JERK 50.0,EXAX_IGN 0}
DECL E6POS XP28={X 680.9328,Y -2572.68799,Z -141.916397,A -67.8898773,B 12.2103901,C 37.8295212,S 2,T 11,E1 4582.3208,E2 0.0,E3 0.0,E4 0.0,E5 0.0,E6 0.0}
DECL FDAT FP28={TOOL_NO 2,BASE_NO 2,IPO_FRAME #BASE,POINT2[] " ",TQ_STATE FALSE}
DECL PDAT PPDAT28={VEL 100.0,ACC 100.0,APO_DIST 100.0,APO_MODE #CDIS}
DECL E6POS XP30={X 1907.59802,Y -7875.57715,Z 2378.80493,A -86.6201935,B -16.2818298,C 91.4838104,S 2,T 11,E1 5636.49512,E2 0.0,E3 0.0,E4 0.0,E5 0.0,E6 0.0}
DECL FDAT FP30={TOOL_NO 2,BASE_NO 0,IPO_FRAME #BASE,POINT2[] " ",TQ_STATE FALSE}
DECL PDAT PPDAT30={VEL 100.0,ACC 100.0,APO_DIST 20.0,APO_MODE #CDIS}
DECL PDAT PPDAT35={VEL 100.0,ACC 100.0,APO_DIST 10.0,APO_MODE #CDIS}
DECL E6POS XP35={X -142.686005,Y -2282.2041,Z 1278.44495,A 13.8204603,B 2.44905901,C -6.20870399,S 2,T 43,E1 1408.61401,E2 0.0,E3 0.0,E4 0.0,E5 0.0,E6 0.0}
DECL FDAT FP35={TOOL_NO 2,BASE_NO 0,IPO_FRAME #BASE,POINT2[] " ",TQ_STATE FALSE}
DECL PDAT PPDAT36={VEL 100.0,ACC 100.0,APO_DIST 5.0,APO_MODE #CDIS}
DECL E6POS XP36={X -694.74707,Y -860.123779,Z 1278.44604,A -105.193901,B 2.44900703,C -6.20870686,S 2,T 42,E1 1408.61401,E2 0.0,E3 0.0,E4 0.0,E5 0.0,E6 0.0}
DECL FDAT FP36={TOOL_NO 2,BASE_NO 0,IPO_FRAME #BASE,POINT2[] " ",TQ_STATE FALSE}
DECL PDAT PPDAT37={VEL 100.0,ACC 100.0,APO_DIST 5.0,APO_MODE #CDIS}
DECL E6POS Xswp_60_0337={X 1321.69104,Y -841.830078,Z 60.7148399,A -3.494941,B 32.0055504,C 89.0259399,S 2,T 11,E1 5553.2749,E2 0.0,E3 0.0,E4 0.0,E5 0.0,E6 0.0}
DECL FDAT Fswp_60_0337={TOOL_NO 2,BASE_NO 2,IPO_FRAME #BASE,POINT2[] " ",TQ_STATE FALSE}
DECL E6POS XP37={X 240.859299,Y 679.959473,Z 1415.14001,A -41.8363991,B 11.3211298,C 18.1852207,S 2,T 2,E1 1820.02405,E2 0.0,E3 0.0,E4 0.0,E5 0.0,E6 0.0}
DECL FDAT FP37={TOOL_NO 2,BASE_NO 0,IPO_FRAME #BASE,POINT2[] " ",TQ_STATE FALSE}
DECL PDAT PPDAT38={VEL 100.0,ACC 100.0,APO_DIST 100.0,APO_MODE #CDIS}
DECL E6POS XP41={X 1435.64795,Y -841.162292,Z 747.776978,A 1.34821701,B -15.5304098,C 91.8447266,S 2,T 11,E1 5636.5,E2 0.0,E3 0.0,E4 0.0,E5 0.0,E6 0.0}
DECL FDAT FP41={TOOL_NO 2,BASE_NO 2,IPO_FRAME #BASE,POINT2[] " ",TQ_STATE FALSE}
DECL PDAT PPDAT42={VEL 100.0,ACC 100.0,APO_DIST 5.0,APO_MODE #CDIS}
DECL E6POS XP42={X 1251.14099,Y -838.862915,Z 486.759308,A 0.970713615,B 46.9011612,C 93.2508469,S 2,T 11,E1 5636.50684,E2 0.0,E3 0.0,E4 0.0,E5 0.0,E6 0.0}
DECL FDAT FP42={TOOL_NO 2,BASE_NO 2,IPO_FRAME #BASE,POINT2[] " ",TQ_STATE FALSE}
DECL PDAT PPDAT43={VEL 100.0,ACC 100.0,APO_DIST 3.0,APO_MODE #CDIS}
DECL E6POS XP43={X 389.176086,Y -1114.28699,Z -102.269798,A 175.624603,B 54.5074883,C -91.0707474,S 2,T 11,E1 4678.20117,E2 0.0,E3 0.0,E4 0.0,E5 0.0,E6 0.0}
DECL FDAT FP43={TOOL_NO 2,BASE_NO 2,IPO_FRAME #BASE,POINT2[] " ",TQ_STATE FALSE}
DECL PDAT PP_OLP84={VEL 100.0,ACC 100.0,APO_DIST 0.0}
DECL E6POS XP47={X -5620.67822,Y -3414.75,Z -364.782715,A -15.1935997,B 2.44905591,C -6.20877123,S 2,T 42,E1 1408.61401,E2 0.0,E3 0.0,E4 0.0,E5 0.0,E6 0.0}
DECL FDAT FP47={TOOL_NO 2,BASE_NO 2,IPO_FRAME #BASE,POINT2[] " ",TQ_STATE FALSE}
DECL PDAT PPDAT51={VEL 100.0,ACC 100.0,APO_DIST 5.0,APO_MODE #CDIS}
DECL PDAT PPDAT55={VEL 100.0,ACC 100.0,APO_DIST 100.0}
DECL PDAT PPDAT56={VEL 100.0,ACC 100.0,APO_DIST 100.0}
DECL PDAT PPDAT57={VEL 100.0,ACC 100.0,APO_DIST 100.0}
DECL PDAT PPDAT58={VEL 100.0,ACC 100.0,APO_DIST 100.0}
DECL E6POS XP50={X 269.843292,Y -848.116577,Z 60.8358002,A -179.496094,B 10.1010799,C -90.1158066,S 2,T 11,E1 4681.69385,E2 0.0,E3 0.0,E4 0.0,E5 0.0,E6 0.0}
DECL FDAT FP50={TOOL_NO 2,BASE_NO 2,IPO_FRAME #BASE,POINT2[] " ",TQ_STATE FALSE}
DECL PDAT PPDAT59={VEL 100.0,ACC 100.0,APO_DIST 10.0,APO_MODE #CDIS}
DECL PDAT PPDAT60={VEL 100.0,ACC 100.0,APO_DIST 100.0}
DECL PDAT PPDAT61={VEL 100.0,ACC 100.0,APO_DIST 100.0}
DECL PDAT PPDAT62={VEL 100.0,ACC 100.0,APO_DIST 100.0}
DECL PDAT PPDAT63={VEL 100.0,ACC 100.0,APO_DIST 100.0}
DECL E6POS XP51={X 278.781891,Y -850.64032,Z 529.158386,A -179.048996,B -22.7865505,C -89.7425766,S 2,T 11,E1 4682.99902,E2 0.0,E3 0.0,E4 0.0,E5 0.0,E6 0.0}
DECL FDAT FP51={TOOL_NO 2,BASE_NO 2,IPO_FRAME #BASE,POINT2[] " ",TQ_STATE FALSE}
DECL PDAT PPDAT65={VEL 100.0,ACC 100.0,APO_DIST 20.0,APO_MODE #CDIS}
DECL E6POS XP53={X 342.528687,Y -1312.19995,Z 567.050598,A 179.099304,B -30.7727299,C -90.2307968,S 2,T 11,E1 4679.25,E2 0.0,E3 0.0,E4 0.0,E5 0.0,E6 0.0}
DECL FDAT FP53={TOOL_NO 2,BASE_NO 2,IPO_FRAME #BASE,POINT2[] " ",TQ_STATE FALSE}
DECL PDAT PPDAT67={VEL 100.0,ACC 100.0,APO_DIST 100.0,APO_MODE #CDIS}
DECL PDAT PPDAT0={VEL 100.0,ACC 100.0,APO_DIST 100.0,APO_MODE #CDIS}
DECL E6POS XP0={X 496.141388,Y -1715.23999,Z -107.852203,A -18.1212292,B -8.07049656,C 74.2473679,S 2,T 11,E1 4684.875,E2 0.0,E3 0.0,E4 0.0,E5 0.0,E6 0.0}
DECL FDAT FP0={TOOL_NO 2,BASE_NO 2,IPO_FRAME #BASE,POINT2[] " ",TQ_STATE FALSE}
DECL PDAT PPDAT69={VEL 100.0,ACC 100.0,APO_DIST 100.0,APO_MODE #CDIS}
DECL E6POS XP55={X -33.49963,Y -879.133728,Z 149.150299,A 18.1609402,B -38.4940681,C 79.5255966,S 2,T 11,E1 4860.08496,E2 0.0,E3 0.0,E4 0.0,E5 0.0,E6 0.0}
DECL FDAT FP55={TOOL_NO 2,BASE_NO 2,IPO_FRAME #BASE,POINT2[] " ",TQ_STATE FALSE}
DECL PDAT PPDAT70={VEL 100.0,ACC 100.0,APO_DIST 30.0,APO_MODE #CDIS}
DECL E6POS XP56={X 99.2140808,Y -846.499817,Z 258.782196,A 18.1166897,B -38.3201714,C 79.6072464,S 2,T 11,E1 4902.61377,E2 0.0,E3 0.0,E4 0.0,E5 0.0,E6 0.0}
DECL FDAT FP56={TOOL_NO 2,BASE_NO 2,IPO_FRAME #BASE,POINT2[] " ",TQ_STATE FALSE}
DECL PDAT PPDAT71={VEL 100.0,ACC 100.0,APO_DIST 100.0,APO_MODE #CDIS}
DECL E6POS XP57={X 107.837502,Y -825.859619,Z 258.730988,A 18.1646595,B -38.4922714,C 79.5321808,S 2,T 11,E1 4907.47314,E2 0.0,E3 0.0,E4 0.0,E5 0.0,E6 0.0}
DECL FDAT FP57={TOOL_NO 2,BASE_NO 2,IPO_FRAME #BASE,POINT2[] " ",TQ_STATE FALSE}
DECL PDAT PP_OLP86={VEL 100.0,ACC 100.0,APO_DIST 0.0}
DECL PDAT PP_OLP87={VEL 100.0,ACC 100.0,APO_DIST 0.0}
DECL PDAT PP_OLP88={VEL 100.0,ACC 100.0,APO_DIST 100.0,APO_MODE #CDIS}
DECL E6POS Xlx788={X 106.594398,Y -825.886902,Z 270.356812,A 18.1619492,B -38.495739,C 79.5243073,S 2,T 11,E1 4905.55518,E2 0.0,E3 0.0,E4 0.0,E5 0.0,E6 0.0}
DECL FDAT Flx788={TOOL_NO 2,BASE_NO 2,IPO_FRAME #BASE,POINT2[] " "}
DECL PDAT PP_OLP89={VEL 100.0,ACC 100.0,APO_DIST 100.0,APO_MODE #CDIS}
DECL E6POS Xlx831={X -33.5169907,Y -895.781006,Z 149.145905,A 18.1617107,B -38.4911385,C 79.5256271,S 2,T 11,E1 4900.61523,E2 0.0,E3 0.0,E4 0.0,E5 0.0,E6 0.0}
DECL FDAT Flx831={TOOL_NO 2,BASE_NO 2,IPO_FRAME #BASE,POINT2[] " "}
DECL E6POS XP59={X 496.141388,Y -1715.23999,Z -107.852203,A -18.1212292,B -8.07049656,C 74.2473679,S 2,T 11,E1 4684.875,E2 0.0,E3 0.0,E4 0.0,E5 0.0,E6 0.0}
DECL FDAT FP59={TOOL_NO 2,BASE_NO 2,IPO_FRAME #BASE,POINT2[] " ",TQ_STATE FALSE}
DECL PDAT PPDAT73={VEL 100.0,ACC 100.0,APO_DIST 100.0,APO_MODE #CDIS}
DECL E6POS XP62={X 390.037506,Y -1524.04297,Z 353.998199,A -179.504196,B 41.2089806,C -87.9716721,S 2,T 11,E1 4687.36084,E2 0.0,E3 0.0,E4 0.0,E5 0.0,E6 0.0}
DECL FDAT FP62={TOOL_NO 2,BASE_NO 2,IPO_FRAME #BASE,POINT2[] " ",TQ_STATE FALSE}
DECL LDAT LCPDAT11={VEL 2.0,ACC 80.0,APO_DIST 20.0,APO_FAC 50.0,AXIS_VEL 100.0,AXIS_ACC 100.0,ORI_TYP #VAR,CIRC_TYP #BASE,JERK_FAC 50.0,GEAR_JERK 50.0,EXAX_IGN 0}
DECL PDAT PPDAT76={VEL 100.0,ACC 100.0,APO_DIST 100.0}
DECL PDAT PP_OLP91={VEL 100.0,ACC 100.0,APO_DIST 0.0}
DECL E6POS Xswp_60_0203={X 258.56131,Y -891.100525,Z 551.157715,A -179.048798,B -22.7876396,C -89.7420273,S 2,T 11,E1 4680.53418,E2 0.0,E3 0.0,E4 0.0,E5 0.0,E6 0.0}
DECL FDAT Fswp_60_0203={TOOL_NO 2,BASE_NO 2,IPO_FRAME #BASE,POINT2[] " "}
DECL PDAT PPDAT77={VEL 100.0,ACC 100.0,APO_DIST 5.0,APO_MODE #CDIS}
DECL E6POS XP63={X 278.777405,Y -824.098328,Z 529.155823,A -179.048904,B -22.7866707,C -89.7424927,S 2,T 11,E1 4679.38281,E2 0.0,E3 0.0,E4 0.0,E5 0.0,E6 0.0}
DECL FDAT FP63={TOOL_NO 2,BASE_NO 2,IPO_FRAME #BASE,POINT2[] " ",TQ_STATE FALSE}
DECL PDAT PPDAT78={VEL 100.0,ACC 100.0,APO_DIST 5.0,APO_MODE #CDIS}
DECL E6POS XP64={X 362.55191,Y -821.745605,Z 567.791321,A 178.825394,B -34.4097099,C -89.7091599,S 2,T 43,E1 4681.0,E2 0.0,E3 0.0,E4 0.0,E5 0.0,E6 0.0}
DECL FDAT FP64={TOOL_NO 2,BASE_NO 2,IPO_FRAME #BASE,POINT2[] " ",TQ_STATE FALSE}
DECL PDAT PPDAT81={VEL 50.0,ACC 100.0,APO_DIST 100.0}
DECL PDAT PPDAT82={VEL 50.0,ACC 100.0,APO_DIST 100.0}
DECL PDAT PPDAT83={VEL 50.0,ACC 100.0,APO_DIST 100.0}
DECL PDAT PPDAT84={VEL 50.0,ACC 100.0,APO_DIST 100.0}
DECL E6POS Xswp_60_0259={X 366.820313,Y -853.075012,Z -120.775597,A 174.980896,B 53.6071014,C -94.6270599,S 2,T 11,E1 4678.04688,E2 0.0,E3 0.0,E4 0.0,E5 0.0,E6 0.0}
DECL FDAT Fswp_60_0259={TOOL_NO 2,BASE_NO 2,IPO_FRAME #BASE,POINT2[] " ",TQ_STATE FALSE}
DECL E6POS Xswp_60_0253={X 259.621399,Y -852.773804,Z -112.924301,A -178.049194,B 45.6860199,C -87.9386673,S 2,T 11,E1 4677.8291,E2 0.0,E3 0.0,E4 0.0,E5 0.0,E6 0.0}
DECL FDAT Fswp_60_0253={TOOL_NO 2,BASE_NO 2,IPO_FRAME #BASE,POINT2[] " ",TQ_STATE FALSE}
DECL E6POS Xswp_60_0249={X 214.160507,Y -853.164429,Z -78.3120117,A -178.291702,B 37.4617691,C -88.298378,S 2,T 11,E1 4677.83301,E2 0.0,E3 0.0,E4 0.0,E5 0.0,E6 0.0}
DECL FDAT Fswp_60_0249={TOOL_NO 2,BASE_NO 2,IPO_FRAME #BASE,POINT2[] " ",TQ_STATE FALSE}
DECL E6POS Xswp_60_0241={X 257.142303,Y -852.976929,Z 45.2910118,A -179.496002,B 10.1006603,C -90.1179733,S 2,T 11,E1 4681.69678,E2 0.0,E3 0.0,E4 0.0,E5 0.0,E6 0.0}
DECL FDAT Fswp_60_0241={TOOL_NO 2,BASE_NO 2,IPO_FRAME #BASE,POINT2[] " ",TQ_STATE FALSE}
DECL E6POS Xswp_60_0239={X 265.541687,Y -851.06073,Z 82.2472382,A -179.690903,B 4.42705202,C -90.1465073,S 2,T 11,E1 4681.69385,E2 0.0,E3 0.0,E4 0.0,E5 0.0,E6 0.0}
DECL FDAT Fswp_60_0239={TOOL_NO 2,BASE_NO 2,IPO_FRAME #BASE,POINT2[] " ",TQ_STATE FALSE}
DECL E6POS Xswp_60_0237={X 262.622711,Y -853.462097,Z 116.181099,A -179.442596,B -10.01577,C -89.6991882,S 2,T 11,E1 4682.28613,E2 0.0,E3 0.0,E4 0.0,E5 0.0,E6 0.0}
DECL FDAT Fswp_60_0237={TOOL_NO 2,BASE_NO 2,IPO_FRAME #BASE,POINT2[] " ",TQ_STATE FALSE}
DECL E6POS Xswp_60_0207={X 222.251907,Y -864.161621,Z 448.493988,A -179.028595,B -7.38161802,C -89.7767029,S 2,T 11,E1 4674.09424,E2 0.0,E3 0.0,E4 0.0,E5 0.0,E6 0.0}
DECL FDAT Fswp_60_0207={TOOL_NO 2,BASE_NO 2,IPO_FRAME #BASE,POINT2[] " ",TQ_STATE FALSE}
DECL E6POS Xswp_60_0211={X 171.578293,Y -861.219177,Z 451.566895,A -175.816406,B -7.38229895,C -89.7748413,S 2,T 11,E1 4674.09082,E2 0.0,E3 0.0,E4 0.0,E5 0.0,E6 0.0}
DECL FDAT Fswp_60_0211={TOOL_NO 2,BASE_NO 2,IPO_FRAME #BASE,POINT2[] " ",TQ_STATE FALSE}
DECL E6POS Xswp_60_0331={X 1214.06104,Y -841.564575,Z 58.9755516,A -1.34586596,B 31.1367798,C 88.9882202,S 2,T 11,E1 5552.93701,E2 0.0,E3 0.0,E4 0.0,E5 0.0,E6 0.0}
DECL FDAT Fswp_60_0331={TOOL_NO 2,BASE_NO 2,IPO_FRAME #BASE,POINT2[] " ",TQ_STATE FALSE}
DECL E6POS Xswp_60_0335={X 1281.28101,Y -841.706726,Z 60.742691,A -3.49542499,B 32.0074692,C 89.0247269,S 2,T 11,E1 5553.27783,E2 0.0,E3 0.0,E4 0.0,E5 0.0,E6 0.0}
DECL FDAT Fswp_60_0335={TOOL_NO 2,BASE_NO 2,IPO_FRAME #BASE,POINT2[] " ",TQ_STATE FALSE}
DECL E6POS Xswp_60_0339={X 1361.61902,Y -841.998718,Z 60.770359,A -3.49538493,B 32.0599518,C 89.028511,S 2,T 11,E1 5553.29883,E2 0.0,E3 0.0,E4 0.0,E5 0.0,E6 0.0}
DECL FDAT Fswp_60_0339={TOOL_NO 2,BASE_NO 2,IPO_FRAME #BASE,POINT2[] " ",TQ_STATE FALSE}
DECL PDAT PPDAT85={VEL 100.0,ACC 80.0,APO_DIST 5.0,APO_MODE #CDIS}
DECL E6POS XPS01010021={X 206.647995,Y -857.749084,Z 303.772003,A -178.132095,B 18.9228992,C -88.8315735,S 2,T 11,E1 4677.62793,E2 0.0,E3 0.0,E4 0.0,E5 0.0,E6 0.0}
DECL FDAT FPS01010021={TOOL_NO 2,BASE_NO 2,IPO_FRAME #BASE,POINT2[] " ",TQ_STATE FALSE}
DECL PDAT PPDAT86={VEL 100.0,ACC 100.0,APO_DIST 100.0}
DECL PDAT PP_OLP15={VEL 100.0,ACC 100.0,APO_DIST 0.0}
DECL E6POS Xswp_60_0396={X 1445.07202,Y -842.604614,Z 678.067871,A 1.23996997,B -7.01102686,C 91.9965591,S 2,T 11,E1 5636.50488,E2 0.0,E3 0.0,E4 0.0,E5 0.0,E6 0.0}
DECL FDAT Fswp_60_0396={TOOL_NO 2,BASE_NO 2,IPO_FRAME #BASE,POINT2[] " "}
DECL E6POS Xswp_60_0397={X 1442.54602,Y -845.039612,Z 712.078186,A 1.29394996,B -11.1452904,C 91.9217529,S 2,T 11,E1 5636.50195,E2 0.0,E3 0.0,E4 0.0,E5 0.0,E6 0.0}
DECL FDAT Fswp_60_0397={TOOL_NO 2,BASE_NO 2,IPO_FRAME #BASE,POINT2[] " ",TQ_STATE FALSE}
DECL PDAT PP_OLP17={VEL 100.0,ACC 100.0,APO_DIST 0.0}
DECL E6POS Xswp_60_0394={X 1475.52795,Y -844.253113,Z 638.954773,A -0.0227528196,B 3.38127303,C 92.2101974,S 2,T 11,E1 5636.49512,E2 0.0,E3 0.0,E4 0.0,E5 0.0,E6 0.0}
DECL FDAT Fswp_60_0394={TOOL_NO 2,BASE_NO 2,IPO_FRAME #BASE,POINT2[] " "}
DECL E6POS Xswp_60_0391={X 1487.88794,Y -844.258911,Z 638.209717,A -0.0223123208,B 3.38131499,C 92.2097168,S 2,T 11,E1 5636.49512,E2 0.0,E3 0.0,E4 0.0,E5 0.0,E6 0.0}
DECL FDAT Fswp_60_0391={TOOL_NO 2,BASE_NO 2,IPO_FRAME #BASE,POINT2[] " ",TQ_STATE FALSE}
ENDDAT
